// TwinCAT 3 PLC project PLC_SortingSystem_PLC
// libraries:
//   Tc2_MC2, * (Beckhoff Automation GmbH)
//   Tc2_Standard, * (Beckhoff Automation GmbH)
//   Tc2_System, * (Beckhoff Automation GmbH)
//   Tc2_Utilities, * (Beckhoff Automation GmbH)
//   Tc3_Module, * (Beckhoff Automation GmbH)
// project tree:
//   01_Submodules/Axis/ FB_Axis.TcPOU
//   01_Submodules/Cylinder/ITFs/ I_Cylinder.TcIO
//   01_Submodules/Cylinder/POUs/ FB_Cylinder.TcPOU, FB_CylinderDiag.TcPOU, FB_CylinderTemp.TcPOU, FB_CylinderTempDiag.TcPOU, FB_CylinderTempRecord.TcPOU
//   01_Submodules/Signal handling/ITFs/ I_SignalHandling.TcIO
//   01_Submodules/Signal handling/POUs/ FB_SignalHandling.TcPOU, FB_SignalHandlingDelay.TcPOU, FB_SignalHandlingIntern.TcPOU
//   02_Subsystems/ E_StateSeparatingAuto.TcDUT, E_StateSortingAutoAxis.TcDUT, E_StateSortingAutoCylinder.TcDUT, FB_SeparatingModule.TcPOU, FB_SortingModule.TcPOU, FB_Subsystem_Root.TcPOU
//   03_Machine/ E_MachineMode.TcDUT, FB_Machine.TcPOU
//   04_Application/ MAIN.TcPOU
//   00_Internal PackAL/DUTs/ E_PMLState.TcDUT, E_PMLUnitMode.TcDUT
//   00_Internal PackAL/POUs/ PS_PackML_StateMachine_Auto.TcPOU, PS_PackML_StateMachine_Maintenance.TcPOU, PS_PackML_StateMachine_Manual.TcPOU, PS_PackML_StateMachine_SemiAuto.TcPOU, PS_UnitModeManager.TcPOU
//   05_Visu/ FB_Visu.TcPOU, GlobalTextList.TcGTLO, Visu_SortingSystem.TcVIS
//   / PlcTask.TcTTO, Visualization Manager.TcVMO (not stored)

CONFIGURATION PLC_SortingSystem_PLC
    RESOURCE PLC ON TwinCAT3
        TASK PlcTask(INTERVAL := T#10ms, PRIORITY := 20);
        PROGRAM MAIN WITH PlcTask : MAIN;
    END_RESOURCE
END_CONFIGURATION

// ---- 02_Subsystems/E_StateSeparatingAuto.TcDUT
{attribute 'qualified_only'}
{attribute 'strict'}
TYPE E_StateSeparatingAuto :
(
	Init := 0,
	Start,
	CloseClamp,
	OpenBarrier,
	CloseBarrier,
	OpenClamp
);
END_TYPE

// ---- 02_Subsystems/E_StateSortingAutoAxis.TcDUT
{attribute 'qualified_only'}
{attribute 'strict'}
TYPE E_StateSortingAutoAxis :
(
	WaitForCylinderAtWorkPos := 0,
	MoveAxis,
	StopAxis
);
END_TYPE

// ---- 02_Subsystems/E_StateSortingAutoCylinder.TcDUT
{attribute 'qualified_only'}
{attribute 'strict'}
TYPE E_StateSortingAutoCylinder :
(
	DetectBox := 0,
	CylToWork,
	CylToBase
);
END_TYPE

// ---- 03_Machine/E_MachineMode.TcDUT
{attribute 'qualified_only'}
{attribute 'strict'}
TYPE E_MachineMode :
(
	Idle := 0,
	Execute := 1,
	Stopped := 2,
	Aborted := 3,
	Starting := 4,
	Stopping := 5,
	Aborting := 6,
	Resetting := 7
);
END_TYPE

// ---- 00_Internal PackAL/DUTs/E_PMLState.TcDUT
(* states according to PackTags v3.0 *)
{attribute 'qualified_only'}
{attribute 'strict'}
TYPE E_PMLState :
(
	UNDEFINED		:=  0,
	CLEARING 		:=  1,
	STOPPED 		:=  2,
	STARTING 		:=  3,
	IDLE 			:=  4,
	SUSPENDED 		:=  5,
	EXECUTE 		:=  6,
	STOPPING	 	:=  7,
	ABORTING 		:=  8,
	ABORTED 		:=  9,
	HOLDING 		:= 10,
	HELD 			:= 11,
	UNHOLDING 		:= 12,
	SUSPENDING 		:= 13,
	UNSUSPENDING 	:= 14,
	RESETTING 		:= 15,
	COMPLETING 		:= 16,
	COMPLETE	 	:= 17
);
END_TYPE

// ---- 00_Internal PackAL/DUTs/E_PMLUnitMode.TcDUT
{attribute 'qualified_only'}
{attribute 'strict'}
TYPE E_PMLUnitMode :
(
	UNDEFINED		:=  0,
	AUTOMATIC		:=  1,
	MAINTENANCE 	:=  2,
	MANUAL 			:=  3,
	SEMIAUTOMATIC	:=  4,
	DRYRUN			:=  5,
	USERMODE1		:=  6,
	USERMODE2		:=  7,
	IDLE 			:=  8,
	ESTOP 			:=  9
);
END_TYPE

// ---- 01_Submodules/Cylinder/ITFs/I_Cylinder.TcIO
INTERFACE I_Cylinder

PROPERTY bState_AtBasePos : BOOL
GET
END_GET
END_PROPERTY

PROPERTY bState_AtWorkPos : BOOL
GET
END_GET
END_PROPERTY

PROPERTY bState_MoveToWork : BOOL
GET
END_GET
END_PROPERTY

METHOD MoveToBase
VAR_INPUT
END_VAR
END_METHOD

METHOD MoveToWork
VAR_INPUT
END_VAR
END_METHOD

METHOD Reset
VAR_INPUT
END_VAR
END_METHOD

END_INTERFACE

// ---- 01_Submodules/Signal handling/ITFs/I_SignalHandling.TcIO
INTERFACE I_SignalHandling

METHOD PUBLIC Enable
VAR_INPUT
	bEnable		: BOOL;
END_VAR
END_METHOD

METHOD SetOutput
VAR_INPUT
END_VAR
END_METHOD

END_INTERFACE

// ---- 04_Application/MAIN.TcPOU
(* =======================================================================================================================================
   OOP: Extended sample
   =======================================================================================================================================
   Description: 
   This PLC sample contains an object-oriented program to control a sorting system.
   The application can be controlled via an integrated visualization.
   
   PLC_SortingSystem_PLC:
   The functionality of the sorting system is implemented within this PLC project (PLC_SortingSystem_PLC).
   It also contains the visualization to control the application.
   
   PLC_SortingSystem_Simu:
   To run the project without hardware, the simulation PLC can be used.
   For example, It simulates the cylinder positions and temperatures, as well as the sensor signals (correspondent to the box positions). 
   =======================================================================================================================================
   InfoSys:
   https://infosys.beckhoff.de/content/1033/tc3_sampleprogram1/45035996374683915.html?id=6126826020926170206
   https://infosys.beckhoff.de/content/1033/tc3_plc_intro/72057596565231755.html?id=3937754078542861062
   ======================================================================================================================================= *)
PROGRAM MAIN
VAR
	fbMachine						: FB_Machine;
	
	//Added Variables
	Plastic_ActPos			AT %Q* 	: LREAL;
	Plastic_ActVelo			AT %Q* 	: LREAL;
	Metal_ActPos			AT %Q* 	: LREAL;
	Metal_ActVelo			AT %Q* 	: LREAL;
	Separating_ActPos		AT %Q* 	: LREAL;
	Separating_ActVelo		AT %Q* 	: LREAL;
	
	{attribute 'TcAnalytics'}
	eMachineState			AT %Q*	: E_MachineMode;
	
	sNetId	: STRING;
	fbGetLocalNetId	:	FB_GetLocalAmsNetId;
	bBusy	: BOOL;
	bInit	: BOOL;
	
	fbConveyorTimerPlastic			: TON;
	fbConveyorTimerMetal			: TON;
	fbConveyorTimerSeparating		: TON;
	tErrorTime						: TIME := T#60M;	
	
END_VAR

// =========================================================

fbMachine();

// =========================================================

Plastic_ActPos := MAIN.fbMachine.fbPlasticSorting.fbAxis.AxisRef.NcToPlc.ActPos;
Plastic_ActVelo := MAIN.fbMachine.fbPlasticSorting.fbAxis.AxisRef.NcToPlc.ActVelo;

Metal_ActPos := MAIN.fbMachine.fbMetalSorting.fbAxis.AxisRef.NcToPlc.ActPos;
Metal_ActVelo := MAIN.fbMachine.fbMetalSorting.fbAxis.AxisRef.NcToPlc.ActVelo;

Separating_ActPos := MAIN.fbMachine.fbSeparateModule.fbAxis.AxisRef.NcToPlc.ActPos;
Separating_ActVelo := MAIN.fbMachine.fbSeparateModule.fbAxis.AxisRef.NcToPlc.ActVelo;

//Handle Conveyor Threshold Overrun
//IF Separating_ActPos > 10000000 THEN
	
//END_IF

//New Machine Enum

IF fbMachine.fbVisu.bIdle THEN
	eMachineState := 0;
ELSIF NOT fbMachine.fbVisu.bButtonPowerIn THEN
	eMachineState := 3;
ELSIF fbMachine.fbVisu.bStarted THEN
	eMachineState := 1;
ELSIF fbMachine.fbVisu.bStopped THEN
	eMachineState := 2;
ELSIF fbMachine.fbVisu.bButtonStartIn THEN
	eMachineState := 4;
ELSIF fbMachine.fbVisu.bButtonStopIn THEN
	eMachineState := 5;
ELSIF fbMachine.fbVisu.bButtonAbortIn THEN
	eMachineState := 6;
ELSIF fbMachine.fbVisu.bReset THEN
	eMachineState := 7;
END_IF

IF NOT bInit THEN
bInit := GetLocalAmsNetId();
END_IF

METHOD GetLocalAmsNetId : BOOL;
VAR_INPUT
END_VAR
fbGetLocalNetId(
	bExecute:= NOT bBusy, 
	bBusy=> bBusy,
	AddrString=> sNetId);
	
IF NOT ((sNetId = '') OR (sNetId = '0.0.0.0.0.0')) THEN
	GetLocalAmsNetId := TRUE;
	RETURN;
END_IF

GetLocalAmsNetId := FALSE;
RETURN;
END_METHOD

END_PROGRAM

// ---- 03_Machine/FB_Machine.TcPOU
FUNCTION_BLOCK FB_Machine
VAR_INPUT
	// =============== Cylinder choice =========================================================
	// Separating module - Clamp cylinder
	bSeparatingClampDiag				: BOOL := TRUE;							// If true the clamp cylinder has diagnosis functionality
	bSeparatingClampTemp				: BOOL := TRUE;							// If true the clamp cylinder has temperature functionality
	bSeparatingClampRecord				: BOOL := FALSE;						// If true the clamp cylinder has recording functionality
	
	// Separating module - Barrier cylinder
	bSeparatingBarrierDiag 				: BOOL := FALSE;						// If true the barrier cylinder has diagnosis functionality
	bSeparatingBarrierTemp 				: BOOL := TRUE;							// If true the barrier cylinder has temperature functionality
	bSeparatingBarrierRecord			: BOOL := TRUE;							// If true the barrier cylinder has recording functionality
	
	// Sorting module for metal boxes - Cylinder
	bMetalSortingCylinderDiag 			: BOOL := TRUE;							// If true the cylinder for metal boxes has diagnosis functionality
	bMetalSortingCylinderTemp 			: BOOL := TRUE;						// If true the cylinder for metal boxes has temperature functionality
	bMetalSortingCylinderRecord 		: BOOL := FALSE;						// If true the cylinder for metal boxes has recording functionality
	
	// Sorting module for plastic boxes - Cylinder
	bPlasticSortingCylinderDiag 		: BOOL := TRUE;							// If true the cylinder for plastic boxes has diagnosis functionality
	bPlasticSortingCylinderTemp 		: BOOL := TRUE;						// If true the cylinder for plastic boxes has temperature functionality
	bPlasticSortingCylinderRecord 		: BOOL := FALSE;						// If true the cylinder for plastic boxes has recording functionality
	

END_VAR
VAR
//
	fbTimerStop						: TON;
	fStopTimePT						: TIME;
	fStartTimePT					: TIME;
	fbTimerStart					: TON;
	fbDRAND							: DRAND;
	fbTon							: TON;
	iTmrET							: INT;
	fRandom							: LREAL;
	bGenerateNumber					: BOOL := TRUE;	
	iDowntimeCounter				: INT;
	fbTimerDowntime					: TON;
	bDowntime						: BOOL;	
	
	// =============== Varying Package Timing ==============================================
	tPackageTime				: TIME;
	fRandValue					: LREAL;
	fbRand						: DRAND;

	// =============== Error ====================================================================
	bError								: BOOL;									// True if modules have errors
	
	// =============== Axis variable ============================================================
	fAxisVelo							: LREAL;								// Axis velocity
	fAxisVeloLastCycle					: LREAL;								// Axis velocity of last cycle
		
	// =============== State machine variables ==================================================
	bStarted							: BOOL;									// True if state machine is in state EXECUTE
	bStopped							: BOOL;									// True if state machine is in state STOPPED
	bReset						AT %Q*	: BOOL;									// True if state machine is in state RESETTING
	bAborted							: BOOL;									// True if state machine is in state ABORTED
	bIdle								: BOOL;									// True if state machine is in state IDLE
	bAuto								: BOOL;									// True if state machine is in mode AUTOMATIC
	bSemi								: BOOL;									// True if state machine is in mode SEMIAUTOMATIC
	bManual								: BOOL;									// True if state machine is in mode MANUAL
	bMaintenance						: BOOL;									// True if state machine is in mode MAINTENANCE
	bStartButtonOff						: BOOL;									// To turn off start button

	// =============== Machine elements =========================================================
	fbSeparateModule					: FB_SeparatingModule;					// Separating module
	fbMetalSorting						: FB_SortingModule;						// Module that sorts metal boxes
	fbPlasticSorting					: FB_SortingModule;						// Module that sorts plastic boxes
	fbComprAir							: FB_SignalHandlingIntern;				// Compressed air
	fbPowerSupply						: FB_SignalHandlingIntern;				// Power supply
	fbVisu								: FB_Visu;								// Visualization

	// =============== Buttons ==================================================================
	fbButtonStart						: FB_SignalHandlingIntern;				// Button to start the machine
	fbButtonStop						: FB_SignalHandlingIntern;				// Button to stop the machine
	fbButtonReset						: FB_SignalHandlingIntern;				// Button to reset the machine
	fbButtonAbort						: FB_SignalHandlingIntern;				// Button to abort the machine
	fbButtonAuto						: FB_SignalHandlingIntern;				// Button to change machine mode to AUTOMATIC
	fbButtonSemi						: FB_SignalHandlingIntern;				// Button to change machine mode to SEMI-AUTOMATIC
	fbButtonManual						: FB_SignalHandlingIntern;				// Button to change machine mode to MANUAL
	fbButtonMaintenance					: FB_SignalHandlingIntern;				// Button to change machine mode to MAINTENANCE
	fbButtonPower						: FB_SignalHandlingIntern;				// Button to control power supply
	fbButtonComprAir					: FB_SignalHandlingIntern;				// Button to control compressed air

	// =============== State machine ============================================================
	fbStateMachineAuto					: PS_PackML_StateMachine_Auto;			// State machine for mode AUTOMATIC
	fbStateMachineSemiAuto				: PS_PackML_StateMachine_SemiAuto;		// State machine for mode SEMI-AUTOMATIC
	fbStateMachineManual				: PS_PackML_StateMachine_Manual;		// State machine for mode MANUAL
	fbStateMachineMaintenance			: PS_PackML_StateMachine_Maintenance;	// State machine for mode MAINTENANCE
	
	ePMLUnitMode						: E_PMLUnitMode := E_PMLUnitMode.IDLE;	// Current mode
	ePMLUnitModeRequested				: E_PMLUnitMode;						// Requested mode
	fbUnitModeManager					: PS_UnitModeManager;					// Mode manager
	ePMLState					AT %Q*	: E_PMLState := E_PMLState.IDLE;			// Current state
	ePMLStateRequested					: E_PMLState;							// Requested state
	
	// =============== Common variables =========================================================
	bInit								: BOOL;									// True if module parameters are initialized
	bAxisEnable							: BOOL;									// True if it is allowed to move axis
	bManualAxisEnable					: BOOL;									// True if it is allowed to move manually axis
	fbTriggerStart						: R_TRIG;								// To diagnose rising edge of start button
	fbTriggerSeparated					: R_TRIG;								// To diagnose rising edge of separated box
	fbTriggerSelectedM					: R_TRIG;								// To diagnose rising edge of selected metal box
	fbTriggerSelectedP					: R_TRIG;								// To diagnose rising edge of selected plastic box
	nBoxesOnTheWay						: INT;									// Number of boxes being moved
	aClampTemps							: ARRAY[1..100] OF LREAL;				// Temperature of clamp cylinder
	aBarrierTemps						: ARRAY[1..100] OF LREAL;				// Temperature of barrier cylinder
	aMetalTemps							: ARRAY[1..100] OF LREAL;				// Temperature of metal cylinder
	aPlasticTemps						: ARRAY[1..100] OF LREAL;				// Temperature of plastic cylinder
	bStartingIsSetToTrue				: BOOL;									// True if the starting methods were called with input TRUE
	bResetIsSetToTrue					: BOOL;									// True if the resetting methods were called with input TRUE
	bHaltIsSetToTrue					: BOOL;									// True if the halting methods were called with input TRUE
	
	cSeparatingBarrierAtWork			: TIME := T#4.5S;									// Time value for separating process: barrier cylinder stays at work position

END_VAR
VAR CONSTANT
	// =============== Axis velocities ==========================================================
	cAxisVeloAutomatic					: LREAL	:= 100.0;						// Axis velocity in (semi) automatic mode
	cAxisVeloNotAutomatic				: LREAL	:= 50.0;						// Axis velocity in non-automatic mode
	
	// =============== Cylinder parameters for separating module (clamp and barrier cylinder) ===
	cSeparatingTimeOutClamp				: TIME 	:= T#2.5S;						// For clamp cylinder with diagnosis: time in which the cylinder should reach base/work position
	cSeparatingRecordIntervalClamp		: TIME 	:= T#1S;						// Time of intervals to record the temperature of clamp cylinder
	cSeparatingTimeOutBarrier			: TIME 	:= T#3S;						// For barrier cylinder with diagnosis: time in which the cylinder should reach base/work position
	cSeparatingRecordIntervalBarrier	: TIME 	:= T#1S;						// Time of intervals to record the temperature of barrier cylinder
	//cSeparatingBarrierAtWork			: TIME 	:= T#4.5S;						// Time value for separating process: barrier cylinder stays at work position
	
	// =============== Cylinder parameters for sorting module ===================================
	cSortingTimeOutCylinder				: TIME 	:= T#3S;						// For sorting cylinder with diagnosis: time in which the cylinder should reach base/work position
	cSortingRecordInterval				: TIME 	:= T#1S;						// Time of intervals to record the temperature of sorting cylinder
	cSortingMoveAxis					: TIME 	:= T#2.5S;						// Time to move sorting axis
	cSortingSensorDelay					: TIME 	:= T#3S;						// Time to delay signal of sorting sensor
END_VAR

// =========================================================
// Getting errors of modules
	
	bError := fbSeparateModule.bAxisError OR fbSeparateModule.bClampError OR fbSeparateModule.bBarrierError
			OR fbMetalSorting.bAxisError OR fbMetalSorting.bCylError 
			OR fbPlasticSorting.bAxisError OR fbPlasticSorting.bCylError;
	
// =========================================================
// Setting velocities of axes

	IF (ePMLUnitMode = E_PMLUnitMode.AUTOMATIC) OR (ePMLUnitMode = E_PMLUnitMode.SEMIAUTOMATIC) THEN
		fAxisVelo := cAxisVeloAutomatic;
	ELSE
		fAxisVelo := cAxisVeloNotAutomatic;
	END_IF

// =========================================================
// Noticing separated and selected boxes
	
	fbTriggerSeparated(CLK := fbSeparateModule.bSeparated);
	fbTriggerSelectedM(CLK := fbMetalSorting.bSelected);
	fbTriggerSelectedP(CLK := fbPlasticSorting.bSelected);
						
// =========================================================
// Getting cylinder temperatures of modules
	
	aBarrierTemps 	:= fbSeparateModule.aBarrierTemps;
	aClampTemps 	:= fbSeparateModule.aClampTemps;
	aMetalTemps 	:= fbMetalSorting.aTemps;
	aPlasticTemps 	:= fbPlasticSorting.aTemps;

// =========================================================
// Cylinder options of modules - choose desired cylinders with more or less functionality
	
	fbSeparateModule.CylinderOptions(	bClampDiag		:= bSeparatingClampDiag, 
										bClampTemp		:= bSeparatingClampTemp, 
										bClampRecord	:= bSeparatingClampRecord, 
										bBarrierDiag	:= bSeparatingBarrierDiag, 
										bBarrierTemp	:= bSeparatingBarrierTemp, 
										bBarrierRecord	:= bSeparatingBarrierRecord);
	
	fbMetalSorting.CylinderOptions(		bCylinderDiag	:= bMetalSortingCylinderDiag,
										bCylinderTemp	:= bMetalSortingCylinderTemp,
										bCylinderRecord	:= bMetalSortingCylinderRecord);
	
	fbPlasticSorting.CylinderOptions(	bCylinderDiag	:= bPlasticSortingCylinderDiag,
										bCylinderTemp	:= bPlasticSortingCylinderTemp,
										bCylinderRecord	:= bPlasticSortingCylinderRecord);

// =========================================================
// Call of actions

	// Init
	General_Init();

	// Mode and state requests
	General_Requests();
	
	// Enable for power supply, compressed air control and buttons
	General_Enable();
	
	// Input variables of separating and sorting modules
	General_ModuleInputs();
	
	// Output variables
	General_SetOutput();
	
	// State machine
	General_StateMachine();
	
	// Visualization
	General_Visu();

// =========================================================
//Timer to Stop Machine/Restart
IF bGenerateNumber THEN
	fbDRAND(Seed:= 0, Num => fRandom);
	bGenerateNumber := FALSE;
END_IF

//Check if machine powered on 
fStartTimePT := LREAL_TO_TIME(fRandom*100000000);
fStopTimePT := LREAL_TO_TIME(fRandom*20000000);

(*IF fbButtonPower.bInput AND NOT bDowntime THEN
	fbTimerStop(IN := NOT fbTimerStart.Q , PT:= fStartTimePT, Q => , ET =>);
	fbTimerStart(IN := fbTimerStop.Q , PT := fStopTimePT, Q =>, ET =>);
	
	IF fbTimerStop.Q AND bStarted THEN
		bGenerateNumber := TRUE;
		fbButtonStop.bInput := TRUE;
		iDowntimeCounter := iDowntimeCounter + 1;
	END_IF
	
	IF fbTimerStart.Q AND bStopped THEN
		bGenerateNumber := TRUE;
		fbButtonStart.bInput := TRUE;	
	END_IF

	IF bIdle THEN
		fbButtonStart.bInput := TRUE;
	END_IF
END_IF

//Implement planned downtime after 10 ON/OFF cycles
IF (iDowntimeCounter > 20) THEN
	fbButtonStop.bInput := TRUE;
	bDowntime := TRUE;
	IF bStopped THEN
	fbButtonPower.bInput := FALSE;
	END_IF	
END_IF

fbTimerDowntime(IN := NOT fbButtonPower.bInput, PT := T#120M, Q =>, ET =>);

IF fbTimerDowntime.Q THEN
	fbButtonPower.bInput := TRUE;
	iDowntimeCounter := 0;
	bDowntime := FALSE;
END_IF

fbRand(Seed:= 0, Num => fRandValue);

tPackageTime := LREAL_TO_TIME((fRandValue*5000) + 5000);

cSeparatingBarrierAtWork := tPackageTime;*)

METHOD PRIVATE General_Enable
VAR_INPUT
END_VAR
// =========================================================
// Power supply

	fbButtonPower.Enable(bEnable := TRUE);
	fbPowerSupply.Enable(bEnable := TRUE);
	
	fbPowerSupply.bInput := fbButtonPower.bOut;

// =========================================================
// Axis control
								
	IF (ePMLState = E_PMLState.ABORTED) THEN
		bAxisEnable := FALSE;
	ELSIF fbPowerSupply.bOut THEN
		bAxisEnable := TRUE;
	END_IF
	
	bManualAxisEnable := fbPowerSupply.bOut AND (ePMLState = E_PMLState.EXECUTE)
						AND ((ePMLUnitMode = E_PMLUnitMode.MANUAL) OR (ePMLUnitMode = E_PMLUnitMode.MAINTENANCE));
						
// =========================================================
// Compressed air control
	
	IF (ePMLUnitMode <> E_PMLUnitMode.MAINTENANCE) THEN
		fbComprAir.bInput := fbPowerSupply.bOut;
	ELSE
		fbComprAir.bInput := fbButtonComprAir.bOut;
	END_IF
	
	fbComprAir.Enable(bEnable := TRUE);
	fbButtonComprAir.Enable(bEnable := (ePMLUnitMode = E_PMLUnitMode.MAINTENANCE));

// =========================================================
// Enable of separate module

	fbSeparateModule.Enable(bComprAirEnabled	:= fbComprAir.bOut,
							bAxisEnable			:= bAxisEnable,
							bSensorEnable		:= TRUE,
							bManualAxisEnable	:= bManualAxisEnable);

// =========================================================
// Enable of sorting module for metal boxes

	fbMetalSorting.Enable(	bComprAirEnabled	:= fbComprAir.bOut,
							bAxisEnable			:= bAxisEnable,
							bSensorEnable		:= TRUE,
							bManualAxisEnable	:= bManualAxisEnable);

// =========================================================
// Enable of sorting module for plastic boxes

	fbPlasticSorting.Enable(bComprAirEnabled	:= fbComprAir.bOut,
							bAxisEnable			:= bAxisEnable,
							bSensorEnable		:= TRUE,
							bManualAxisEnable	:= bManualAxisEnable);

// =========================================================
// States and modes
		
	// Start button
	fbButtonStart.Enable(bEnable		:= NOT ((ePMLState = E_PMLState.IDLE) AND bError));
	
	// Stop button
	fbButtonStop.Enable(bEnable 		:= (ePMLState = E_PMLState.STOPPING) OR (ePMLState = E_PMLState.EXECUTE) OR (ePMLState = E_PMLState.IDLE));
	
	// Reset button
	fbButtonReset.Enable(bEnable		:= (ePMLState = E_PMLState.STOPPED));
	
	// Abort button
	fbButtonAbort.bInput 				:= NOT fbPowerSupply.bOut;
	
	fbButtonAbort.Enable(bEnable 		:= (ePMLState = E_PMLState.EXECUTE) OR (ePMLState = E_PMLState.STOPPING) OR (ePMLState = E_PMLState.RESETTING));
								
	// Automatic mode button
	fbButtonAuto.Enable(bEnable 		:= (ePMLState = E_PMLState.IDLE) AND (ePMLUnitMode <> E_PMLUnitMode.AUTOMATIC));
	
	// Semi-automatic mode button
	fbButtonSemi.Enable(bEnable 		:= (ePMLState = E_PMLState.IDLE) AND (ePMLUnitMode <> E_PMLUnitMode.SEMIAUTOMATIC));
	
	// Manual mode button
	fbButtonManual.Enable(bEnable 		:= (ePMLState = E_PMLState.IDLE) AND (ePMLUnitMode <> E_PMLUnitMode.MANUAL));
	
	// Maintenance mode button
	fbButtonMaintenance.Enable(bEnable	:= (ePMLState = E_PMLState.IDLE) AND (ePMLUnitMode <> E_PMLUnitMode.MAINTENANCE));

// =========================================================
END_METHOD

METHOD PRIVATE General_Init
VAR_INPUT
END_VAR
// =========================================================

IF NOT bInit THEN
	
	// Time values of separating module
		// Clamp cylinder
		fbSeparateModule.tTimeOutOfClamp 			:= cSeparatingTimeOutClamp;
		fbSeparateModule.tRecordIntervalOfClamp		:= cSeparatingRecordIntervalClamp;
		
		// Barrier cylinder
		fbSeparateModule.tTimeOutOfBarrier 			:= cSeparatingTimeOutBarrier;
		fbSeparateModule.tRecordIntervalOfBarrier 	:= cSeparatingRecordIntervalBarrier;
		
		// Separating process
		fbSeparateModule.tBarrierAtWorkPos				:= cSeparatingBarrierAtWork;

	// Time values of sorting module (metal boxes)
		fbMetalSorting.tTimeOutOfCylinder 			:= cSortingTimeOutCylinder;
		fbMetalSorting.tRecordIntervalOfCylinder 	:= cSortingRecordInterval;
		fbMetalSorting.tAxisMovement 				:= cSortingMoveAxis;
		fbMetalSorting.tDelayOfSensor 				:= cSortingSensorDelay;
		
	// Time values of sorting module (plastic boxes)
		fbPlasticSorting.tTimeOutOfCylinder 		:= cSortingTimeOutCylinder;
		fbPlasticSorting.tRecordIntervalOfCylinder := cSortingRecordInterval;
		fbPlasticSorting.tAxisMovement 				:= cSortingMoveAxis;
		fbPlasticSorting.tDelayOfSensor 			:= cSortingSensorDelay;

	// Init done
		bInit := TRUE;
END_IF

// =========================================================
END_METHOD

METHOD PRIVATE General_ModuleInputs
VAR_INPUT
END_VAR
// =========================================================
// Separating modul

	// Sate and button signals
	fbSeparateModule.bExecute 			:= (ePMLState = E_PMLState.EXECUTE);
	fbSeparateModule.bSemiStart 		:= fbTriggerStart.Q;
	
	// Axis velocity has changed
	IF (fAxisVeloLastCycle <> fAxisVelo) THEN
		fbSeparateModule.fAxisVelocity 	:= fAxisVelo;
	END_IF
	
	// Information about number of boxes being sorted
	fbSeparateModule.nBoxesOnTheWay 	:= nBoxesOnTheWay;

// =========================================================
// Sorting modul for metal boxes
	
	// Axis velocity has changed
	IF (fAxisVeloLastCycle <> fAxisVelo) THEN
		fbMetalSorting.fAxisVelocity 	:= fAxisVelo;
	END_IF

// =========================================================
// Sorting modul for plastic boxes

	// Axis velocity has changed
	IF (fAxisVeloLastCycle <> fAxisVelo) THEN
		fbPlasticSorting.fAxisVelocity 	:= fAxisVelo;
	END_IF
	
// =========================================================
/// Remember axis velocity of this cycle for next cycle => call of property AxisVelocity is event triggered

	fAxisVeloLastCycle := fAxisVelo;

// =========================================================
END_METHOD

METHOD PRIVATE General_Requests
VAR_INPUT
END_VAR
// =========================================================
// Check for state requests

	fbTriggerStart( CLK := fbButtonStart.bOut);
	
	IF bStartButtonOff AND NOT fbButtonStart.bInput THEN
		bStartButtonOff := FALSE;
	END_IF
	
	IF fbTriggerStart.Q THEN
		bStartButtonOff := TRUE;
	
		IF ePMLState = E_PMLState.ABORTED THEN
			ePMLStateRequested := E_PMLState.CLEARING;
			
		ELSIF ePMLState = E_PMLState.STOPPED THEN
			ePMLStateRequested := E_PMLState.RESETTING;
			
		ELSIF ePMLState = E_PMLState.IDLE AND fbPowerSupply.bOut THEN
			ePMLStateRequested := E_PMLState.STARTING;
		END_IF
		
	ELSIF fbButtonStop.bOut THEN
		ePMLStateRequested := E_PMLState.STOPPING;
		
	ELSIF fbButtonReset.bOut THEN
		ePMLStateRequested := E_PMLState.RESETTING;
	END_IF

// =========================================================
// Check for mode requests

	IF fbButtonManual.bOut THEN
		ePMLUnitModeRequested := E_PMLUnitMode.MANUAL;
		
	ELSIF fbButtonAuto.bOut THEN
		ePMLUnitModeRequested := E_PMLUnitMode.AUTOMATIC;
		
	ELSIF fbButtonSemi.bOut THEN
		ePMLUnitModeRequested := E_PMLUnitMode.SEMIAUTOMATIC;
		
	ELSIF fbButtonMaintenance.bOut THEN
		ePMLUnitModeRequested := E_PMLUnitMode.MAINTENANCE;
	END_IF
	
	IF fbButtonManual.bOut OR fbButtonAuto.bOut OR fbButtonSemi.bOut OR fbButtonMaintenance.bOut THEN
		fbUnitModeManager(	Execute 		:= TRUE,
							eModeCommand 	:= ePMLUnitModeRequested,
							ePMLState 		:= ePMLState);
	END_IF
	
	IF fbUnitModeManager.Done THEN
		ePMLUnitMode := fbUnitModeManager.eModeStatus;
		
		fbUnitModeManager(Execute := FALSE);
	END_IF
	
// =========================================================
END_METHOD

METHOD PRIVATE General_SetOutput
VAR_INPUT
END_VAR
// =========================================================
// State variables

	bStopped 		:= (ePMLState = E_PMLState.STOPPED);
	bStarted 		:= (ePMLState = E_PMLState.EXECUTE);
	bReset 			:= (ePMLState = E_PMLState.RESETTING);
	bAborted 		:= (ePMLState = E_PMLState.ABORTED);
	bIdle 			:= (ePMLState = E_PMLState.IDLE AND fbPowerSupply.bOut);

// =========================================================
// Mode variables

	bAuto 			:= (ePMLUnitMode = E_PMLUnitMode.AUTOMATIC);
	bSemi 			:= (ePMLUnitMode = E_PMLUnitMode.SEMIAUTOMATIC);
	bManual 		:= (ePMLUnitMode = E_PMLUnitMode.MANUAL);
	bMaintenance 	:= (ePMLUnitMode = E_PMLUnitMode.MAINTENANCE);

// =========================================================
// Power supply and compressed air control
		
	fbPowerSupply.SetOutput();
	fbComprAir.SetOutput();		

// =========================================================
// Modules

	fbSeparateModule.InputOutput();
	fbMetalSorting.InputOutput();
	fbPlasticSorting.InputOutput();

// =========================================================
// Buttons

	// Power supply and compressed air control
	fbButtonPower.SetOutput();
	fbButtonComprAir.SetOutput();	
	
	// States
	fbButtonStart.SetOutput();
	fbButtonStop.SetOutput();
	fbButtonReset.SetOutput();
	fbButtonAbort.SetOutput();
	
	// Modes
	fbButtonAuto.SetOutput();
	fbButtonSemi.SetOutput();
	fbButtonManual.SetOutput();
	fbButtonMaintenance.SetOutput();	
	
// =========================================================
END_METHOD

METHOD PRIVATE General_StateMachine
VAR_INPUT
END_VAR
// =========================================================
	// Mode and state handling
	
CASE ePMLUnitMode OF
	
	// =========================================================	
	E_PMLUnitMode.AUTOMATIC:		

				fbStateMachineAuto(	Start 	:= ePMLStateRequested = E_PMLState.STARTING,
									Stop 	:= fbButtonStop.bOut,
									Reset 	:= fbButtonReset.bOut OR ePMLStateRequested = E_PMLState.RESETTING,
									Clear 	:= ePMLStateRequested = E_PMLState.CLEARING,
									Abort 	:= fbButtonAbort.bOut OR (bError AND ePMLState = E_PMLState.EXECUTE));
								 
				ePMLState := fbStateMachineAuto.ePMLState;
				
				Operating_Automatic();

	// =========================================================	
	E_PMLUnitMode.MANUAL:		

				fbStateMachineManual(	Start 	:= ePMLStateRequested = E_PMLState.STARTING,
										Stop 	:= fbButtonStop.bOut,
										Reset 	:= fbButtonReset.bOut OR ePMLStateRequested = E_PMLState.RESETTING,
										Clear 	:= ePMLStateRequested = E_PMLState.CLEARING,
										Abort 	:= fbButtonAbort.bOut OR (bError AND ePMLState = E_PMLState.EXECUTE));
									 
				ePMLState := fbStateMachineManual.ePMLState;
				
				Operating_Manual();
	
	// =========================================================						
	E_PMLUnitMode.SEMIAUTOMATIC:	

				fbStateMachineSemiAuto(	Start 	:= ePMLStateRequested = E_PMLState.STARTING,
									 	Stop 	:= fbButtonStop.bOut,
										Reset 	:= fbButtonReset.bOut OR ePMLStateRequested = E_PMLState.RESETTING,
										Clear 	:= ePMLStateRequested = E_PMLState.CLEARING,
										Abort 	:= fbButtonAbort.bOut OR (bError AND ePMLState = E_PMLState.EXECUTE));
									 
				ePMLState := fbStateMachineSemiAuto.ePMLState;
				
				Operating_Semiautomatic();
	
	// =========================================================						
	E_PMLUnitMode.MAINTENANCE:	

				fbStateMachineMaintenance(	Start 	:= ePMLStateRequested = E_PMLState.STARTING,
											Stop 	:= fbButtonStop.bOut,
											Reset 	:= fbButtonReset.bOut OR ePMLStateRequested = E_PMLState.RESETTING,
											Clear 	:= ePMLStateRequested = E_PMLState.CLEARING,
											Abort 	:= fbButtonAbort.bOut OR (bError AND ePMLState = E_PMLState.EXECUTE));
									 
				ePMLState := fbStateMachineMaintenance.ePMLState;
				
				Operating_Maintenance();
END_CASE

// =========================================================
END_METHOD

METHOD PRIVATE General_Visu
VAR_INPUT
END_VAR
// =========================================================
		// Calling visu function block
		
fbVisu(	bError  				:= bError, 
		fAxisVelo 				:= fAxisVelo, 
		bComprAirEnabled 		:= fbComprAir.bOut, 
		bPowerEnabled 			:= fbPowerSupply.bOut, 
		bMainAxisMoves 			:= fbSeparateModule.bAxisMoves, 
		bMetalAxisMoves 		:= fbMetalSorting.bAxisMoves, 
		bPlasticAxisMoves 		:= fbPlasticSorting.bAxisMoves, 
		bClampToWork 			:= fbSeparateModule.bClampToWork, 
		bBarrierToWork 			:= fbSeparateModule.bBarrierToWork, 
		bMetalToWork 			:= fbMetalSorting.bCylinderToWork, 
		bPlasticToWork 			:= fbPlasticSorting.bCylinderToWork, 
		bClampError 			:= fbSeparateModule.bClampError, 
		sClampErrMsg 			:= fbSeparateModule.sClampErrorMsg, 
		bMetalCylError 			:= fbMetalSorting.bCylError, 
		sMetalErrMsg 			:= fbMetalSorting.sCylErrorMsg, 
		bPlasticCylError 		:= fbPlasticSorting.bCylError, 
		sPlasticErrMsg 			:= fbPlasticSorting.sCylErrorMsg, 
		nMainAxisErrorId 		:= fbSeparateModule.fbAxis.nErrorID, 
		nMetalAxisErrorId 		:= fbMetalSorting.fbAxis.nErrorID, 
		nPlasticAxisErrorId		:= fbPlasticSorting.fbAxis.nErrorID, 
		bStarted 				:= bStarted, 
		bStopped 				:= bStopped, 
		bReset 					:= bReset, 
		bAborted 				:= bAborted, 
		bIdle					:= bIdle, 
		bAuto 					:= bAuto, 
		bSemi 					:= bSemi, 
		bManual 				:= bManual, 
		bMaintenance 			:= bMaintenance, 
		bStartButtonOff 		:= bStartButtonOff, 
		bButtonPowerIn 			:= fbButtonPower.bOut, 
		bButtonComprAirIn 		:= fbButtonComprAir.bOut, 
		bButtonStartIn 			:= fbButtonStart.bOut, 
		bButtonStopIn 			:= fbButtonStop.bOut, 
		bButtonResetIn 			:= fbButtonReset.bOut, 
		bButtonAbortIn 			:= fbButtonAbort.bOut, 
		bButtonAutoIn 			:= fbButtonAuto.bOut, 
		bButtonSemiIn 			:= fbButtonSemi.bOut, 
		bButtonManuIn 			:= fbButtonManual.bOut, 
		bButtonMaintenanceIn 	:= fbButtonMaintenance.bOut, 
		bButtonMainFwIn 		:= fbSeparateModule.bButtonAxisFwOut,
		bButtonMainBwIn 		:= fbSeparateModule.bButtonAxisBwOut, 
		bButtonMetalFwIn 		:= fbMetalSorting.bButtonAxisFwOut, 
		bButtonMetalBwIn 		:= fbMetalSorting.bButtonAxisBwOut, 
		bButtonPlasticFwIn 		:= fbPlasticSorting.bButtonAxisFwOut, 
		bButtonPlasticBwIn 		:= fbPlasticSorting.bButtonAxisBwOut, 
		bButtonClampToWorkIn 	:= fbSeparateModule.bButtonClampToWorkOut, 
		bButtonBarrierToWorkIn 	:= fbSeparateModule.bButtonBarrierToWorkOut, 
		bButtonMetalToWorkIn 	:= fbMetalSorting.bButtonCylToWorkOut, 
		bButtonPlasticToWorkIn 	:= fbPlasticSorting.bButtonCylToWorkOut, 
		
		bButtonPowerOut			=> fbButtonPower.bInput, 
		bButtonComprAirOut 		=> fbButtonComprAir.bInput, 
		bButtonStartOut 		=> fbButtonStart.bInput, 
		bButtonStopOut 			=> fbButtonStop.bInput, 
		bButtonResetOut 		=> fbButtonReset.bInput, 
		bButtonAutoOut 			=> fbButtonAuto.bInput, 
		bButtonSemiOut 			=> fbButtonSemi.bInput, 
		bButtonManuOut 			=> fbButtonManual.bInput, 
		bButtonMaintenanceOut 	=> fbButtonMaintenance.bInput, 
		bButtonMainFwOut 		=> fbSeparateModule.bButtonAxisFwIn, 
		bButtonMainBwOut 		=> fbSeparateModule.bButtonAxisBwIn, 
		bButtonMetalFwOut 		=> fbMetalSorting.bButtonAxisFwIn, 
		bButtonMetalBwOut 		=> fbMetalSorting.bButtonAxisBwIn, 
		bButtonPlasticFwOut		=> fbPlasticSorting.bButtonAxisFwIn, 
		bButtonPlasticBwOut		=> fbPlasticSorting.bButtonAxisBwIn, 
		bButtonClampToWorkOut 	=> fbSeparateModule.bButtonClampToWorkIn, 
		bButtonBarrierToWorkOut	=> fbSeparateModule.bButtonBarrierToWorkIn, 
		bButtonMetalToWorkOut 	=> fbMetalSorting.bButtonCylToWorkIn, 
		bButtonPlasticToWorkOut	=> fbPlasticSorting.bButtonCylToWorkIn);
	
// =========================================================
END_METHOD

METHOD PRIVATE Operating_Automatic
VAR_INPUT
END_VAR
// =========================================================

CASE ePMLState OF
	
	// =========================================================
	// Turning axis reset off, passing it to axis instances
	E_PMLState.IDLE:
	
				IF bResetIsSetToTrue THEN
					bResetIsSetToTrue := FALSE;
					
					fbSeparateModule.Reset(bReset := FALSE);							
					fbMetalSorting.Reset(bReset := FALSE);
					fbPlasticSorting.Reset(bReset := FALSE);
					
					fbStateMachineAuto.StateComplete := FALSE;	
				END_IF
	
	// =========================================================
	// Resetting variables for executing automatic mode, checking status of axes
	E_PMLState.STARTING:
	
				IF NOT bStartingIsSetToTrue THEN
					bStartingIsSetToTrue := TRUE;
					
					fbSeparateModule.Starting(bStarting := TRUE);
					fbMetalSorting.Starting(bStarting := TRUE);
					fbPlasticSorting.Starting(bStarting := TRUE);
				END_IF

				IF NOT fbSeparateModule.bState_StartingDone THEN
					fbSeparateModule.Starting(bStarting := TRUE);
				END_IF
				
				IF NOT fbMetalSorting.bState_StartingDone THEN
					fbMetalSorting.Starting(bStarting := TRUE);
				END_IF
				
				IF NOT fbPlasticSorting.bState_StartingDone THEN
					fbPlasticSorting.Starting(bStarting := TRUE);
				END_IF

				IF fbSeparateModule.bState_StartingDone AND fbMetalSorting.bState_StartingDone AND fbPlasticSorting.bState_StartingDone THEN
					fbStateMachineAuto.StateComplete := TRUE;
				END_IF

	// =========================================================
	// Executing automatic mode
	E_PMLState.EXECUTE:	

				IF bStartingIsSetToTrue THEN
					bStartingIsSetToTrue := FALSE;
					
					fbSeparateModule.Starting(bStarting := FALSE);
					fbMetalSorting.Starting(bStarting := FALSE);	
					fbPlasticSorting.Starting(bStarting := FALSE);
					
					fbStateMachineAuto.StateComplete := FALSE;
				END_IF
				
				fbSeparateModule.Automatic();
				fbMetalSorting.Automatic();
				fbPlasticSorting.Automatic();
				
				IF fbTriggerSeparated.Q THEN
					nBoxesOnTheWay := nBoxesOnTheWay + 1;
				END_IF
				
				IF fbTriggerSelectedM.Q THEN
					nBoxesOnTheWay := nBoxesOnTheWay - 1;
				END_IF
				
				IF fbTriggerSelectedP.Q THEN
					nBoxesOnTheWay := nBoxesOnTheWay - 1;
				END_IF
						
	// =========================================================
	// Stopping axes
	E_PMLState.ABORTING:

				IF NOT bHaltIsSetToTrue THEN
					bHaltIsSetToTrue := TRUE;
					
					fbSeparateModule.Stop(bHalt := TRUE);
					fbMetalSorting.Stop(bHalt := TRUE);
					fbPlasticSorting.Stop(bHalt := TRUE);
				END_IF

				IF NOT fbSeparateModule.bState_HaltDone THEN
					fbSeparateModule.Stop(bHalt := TRUE);
				END_IF
				
				IF NOT fbMetalSorting.bState_HaltDone THEN
					fbMetalSorting.Stop(bHalt := TRUE);
				END_IF
				
				IF NOT fbPlasticSorting.bState_HaltDone THEN
					fbPlasticSorting.Stop(bHalt := TRUE);
				END_IF

				IF fbSeparateModule.bState_HaltDone AND fbMetalSorting.bState_HaltDone AND fbPlasticSorting.bState_HaltDone THEN
					fbStateMachineAuto.StateComplete := TRUE;
				END_IF
	
	// =========================================================
	// Turning off axis stop, passing it to axis instances
	E_PMLState.ABORTED:
				
				IF bHaltIsSetToTrue THEN
					bHaltIsSetToTrue := FALSE;
					
					fbSeparateModule.Stop(bHalt := FALSE);
					fbMetalSorting.Stop(bHalt := FALSE);
					fbPlasticSorting.Stop(bHalt := FALSE);
				END_IF
				
				IF fbStateMachineAuto.StateComplete THEN
					fbStateMachineAuto.StateComplete := FALSE;
				END_IF
	
	// =========================================================
	E_PMLState.CLEARING:

				fbStateMachineAuto.StateComplete := TRUE;
	
	// =========================================================
	// Selecting boxes on conveyor belt to destination, then stopping axes
	E_PMLState.STOPPING:	

				IF fbTriggerSeparated.Q THEN
					nBoxesOnTheWay := nBoxesOnTheWay + 1;
				END_IF
				
				IF fbTriggerSelectedM.Q THEN
					nBoxesOnTheWay := nBoxesOnTheWay - 1;
				END_IF
				
				IF fbTriggerSelectedP.Q THEN
					nBoxesOnTheWay := nBoxesOnTheWay - 1;
				END_IF
				
				IF (nBoxesOnTheWay = 0) AND NOT bHaltIsSetToTrue THEN
					bHaltIsSetToTrue := TRUE;
		
					fbSeparateModule.Stop(bHalt := TRUE);				
					fbMetalSorting.Stop(bHalt := TRUE);				
					fbPlasticSorting.Stop(bHalt := TRUE);			
				END_IF
				
				IF NOT fbSeparateModule.bState_HaltDone OR (nBoxesOnTheWay <> 0) THEN
					fbSeparateModule.Automatic();
					
					IF (nBoxesOnTheWay = 0) THEN
						fbSeparateModule.Stop(bHalt := TRUE);
					END_IF
				END_IF
				
				IF NOT fbMetalSorting.bState_HaltDone OR (nBoxesOnTheWay <> 0) THEN
					fbMetalSorting.Automatic();
					
					IF (nBoxesOnTheWay = 0) THEN
						fbMetalSorting.Stop(bHalt := TRUE);
					END_IF
				END_IF
				
				IF NOT fbPlasticSorting.bState_HaltDone OR (nBoxesOnTheWay <> 0) THEN
					fbPlasticSorting.Automatic();
					
					IF (nBoxesOnTheWay = 0) THEN
						fbPlasticSorting.Stop(bHalt := TRUE);
					END_IF
				END_IF

				IF fbSeparateModule.bState_HaltDone AND fbMetalSorting.bState_HaltDone
				AND fbPlasticSorting.bState_HaltDone AND (nBoxesOnTheWay = 0) THEN
					fbStateMachineAuto.StateComplete := TRUE;
				END_IF
					
	// =========================================================
	// Turning off axis stop, passing it to axis instances
	E_PMLState.STOPPED:	

				IF bHaltIsSetToTrue THEN
					bHaltIsSetToTrue := FALSE;
					
					fbSeparateModule.Stop(bHalt := FALSE);	
					fbMetalSorting.Stop(bHalt := FALSE);			
					fbPlasticSorting.Stop(bHalt := FALSE);
				END_IF

				IF fbStateMachineAuto.StateComplete THEN
					fbStateMachineAuto.StateComplete := FALSE;	
				END_IF

	// =========================================================
	// Resetting cylinders and axes
	E_PMLState.RESETTING:	

				IF NOT bResetIsSetToTrue THEN
					bResetIsSetToTrue := TRUE;
					
					fbSeparateModule.Reset(bReset := TRUE);							
					fbMetalSorting.Reset(bReset := TRUE);
					fbPlasticSorting.Reset(bReset := TRUE);
				END_IF
				
				IF NOT fbSeparateModule.bState_ResetDone THEN
					fbSeparateModule.Reset(bReset := TRUE);
				END_IF
				
				IF NOT fbMetalSorting.bState_ResetDone THEN
					fbMetalSorting.Reset(bReset := TRUE);
				END_IF
				
				IF NOT fbPlasticSorting.bState_ResetDone THEN
					fbPlasticSorting.Reset(bReset := TRUE);
				END_IF
				
				IF fbSeparateModule.bState_ResetDone AND fbMetalSorting.bState_ResetDone AND fbPlasticSorting.bState_ResetDone 
				AND fbSeparateModule.bState_ClampAtBasePos AND fbSeparateModule.bState_BarrierAtBasePos
				AND fbMetalSorting.bState_CylinderAtBasePos AND fbPlasticSorting.bState_CylinderAtBasePos THEN
					nBoxesOnTheWay 						:= 0;
					fbStateMachineAuto.StateComplete 	:= TRUE;
				END_IF
END_CASE

// =========================================================
END_METHOD

METHOD PRIVATE Operating_Maintenance
VAR_INPUT
END_VAR
// =========================================================

CASE ePMLState OF
	
	// =========================================================
	// Turning axis reset off, passing it to axis instances
	E_PMLState.IDLE:		

				IF bResetIsSetToTrue THEN
					bResetIsSetToTrue := FALSE;
					
					fbSeparateModule.Reset(bReset := FALSE);
					fbMetalSorting.Reset(bReset := FALSE);
					fbPlasticSorting.Reset(bReset := FALSE);
					
					fbStateMachineMaintenance.StateComplete := FALSE;
				END_IF
	
	// =========================================================
	// Checking status of axes
	E_PMLState.STARTING:	

				IF NOT bStartingIsSetToTrue THEN
					bStartingIsSetToTrue := TRUE;
					
					fbSeparateModule.Starting(bStarting := TRUE);
					fbMetalSorting.Starting(bStarting := TRUE);
					fbPlasticSorting.Starting(bStarting := TRUE);
				END_IF

				IF NOT fbSeparateModule.bState_StartingDone THEN
					fbSeparateModule.Starting(bStarting := TRUE);
				END_IF
				
				IF NOT fbMetalSorting.bState_StartingDone THEN
					fbMetalSorting.Starting(bStarting := TRUE);
				END_IF
				
				IF NOT fbPlasticSorting.bState_StartingDone THEN
					fbPlasticSorting.Starting(bStarting := TRUE);
				END_IF

				IF fbSeparateModule.bState_StartingDone AND fbMetalSorting.bState_StartingDone AND fbPlasticSorting.bState_StartingDone THEN
					fbStateMachineMaintenance.StateComplete := TRUE;
				END_IF

	// =========================================================
	// Executing maintenance mode
	E_PMLState.EXECUTE:	

				IF bStartingIsSetToTrue THEN
					bStartingIsSetToTrue := FALSE;
					
					fbSeparateModule.Starting(bStarting := FALSE);
					fbMetalSorting.Starting(bStarting := FALSE);	
					fbPlasticSorting.Starting(bStarting := FALSE);
					
					fbStateMachineMaintenance.StateComplete := FALSE;
				END_IF
				
				fbSeparateModule.Maintenance();
				fbMetalSorting.Maintenance();
				fbPlasticSorting.Maintenance();
						
	// =========================================================
	// Stopping axes
	E_PMLState.ABORTING:	

				IF NOT bHaltIsSetToTrue THEN
					bHaltIsSetToTrue := TRUE;
					
					fbSeparateModule.Stop(bHalt := TRUE);
					fbMetalSorting.Stop(bHalt := TRUE);
					fbPlasticSorting.Stop(bHalt := TRUE);
				END_IF

				IF NOT fbSeparateModule.bState_HaltDone THEN
					fbSeparateModule.Stop(bHalt := TRUE);
				END_IF
				
				IF NOT fbMetalSorting.bState_HaltDone THEN
					fbMetalSorting.Stop(bHalt := TRUE);
				END_IF
				
				IF NOT fbPlasticSorting.bState_HaltDone THEN
					fbPlasticSorting.Stop(bHalt := TRUE);
				END_IF

				IF fbSeparateModule.bState_HaltDone AND fbMetalSorting.bState_HaltDone AND fbPlasticSorting.bState_HaltDone THEN
					fbStateMachineMaintenance.StateComplete := TRUE;
				END_IF
	
	// =========================================================
	// Turning off axis stop, passing it to axis instances
	E_PMLState.ABORTED:	

				IF bHaltIsSetToTrue THEN
					bHaltIsSetToTrue := FALSE;
					
					fbSeparateModule.Stop(bHalt := FALSE);
					fbMetalSorting.Stop(bHalt := FALSE);
					fbPlasticSorting.Stop(bHalt := FALSE);
				END_IF

				IF fbStateMachineMaintenance.StateComplete THEN
					fbStateMachineMaintenance.StateComplete := FALSE;
				END_IF
	
	// =========================================================
	E_PMLState.CLEARING:	

				fbStateMachineMaintenance.StateComplete := TRUE;
	
	// =========================================================
	// Stopping axes
	E_PMLState.STOPPING:	

				IF NOT bHaltIsSetToTrue THEN
					bHaltIsSetToTrue := TRUE;

					fbSeparateModule.Stop(bHalt := TRUE);				
					fbMetalSorting.Stop(bHalt := TRUE);				
					fbPlasticSorting.Stop(bHalt := TRUE);				
				END_IF

				IF NOT fbSeparateModule.bState_HaltDone THEN
					fbSeparateModule.Stop(bHalt := TRUE);
				END_IF
				
				IF NOT fbMetalSorting.bState_HaltDone THEN
					fbMetalSorting.Stop(bHalt := TRUE);
				END_IF
				
				IF NOT fbPlasticSorting.bState_HaltDone THEN
					fbPlasticSorting.Stop(bHalt := TRUE);
				END_IF

				IF fbSeparateModule.bState_HaltDone AND fbMetalSorting.bState_HaltDone AND fbPlasticSorting.bState_HaltDone THEN
						fbStateMachineMaintenance.StateComplete := TRUE;
				END_IF
					
	// =========================================================
	// Turning off axis stop, passing it to axis instances
	E_PMLState.STOPPED:	

				IF bHaltIsSetToTrue THEN
					bHaltIsSetToTrue := FALSE;
					
					fbSeparateModule.Stop(bHalt := FALSE);	
					fbMetalSorting.Stop(bHalt := FALSE);			
					fbPlasticSorting.Stop(bHalt := FALSE);
				END_IF

				IF fbStateMachineMaintenance.StateComplete THEN
					fbStateMachineMaintenance.StateComplete := FALSE;
				END_IF

	// =========================================================
	// Resetting cylinders and axes
	E_PMLState.RESETTING:	

				IF NOT bResetIsSetToTrue THEN
					bResetIsSetToTrue := TRUE;
					
					fbSeparateModule.Reset(bReset := TRUE);							
					fbMetalSorting.Reset(bReset := TRUE);
					fbPlasticSorting.Reset(bReset := TRUE);
				END_IF
				
				IF NOT fbSeparateModule.bState_ResetDone THEN
					fbSeparateModule.Reset(bReset := TRUE);
				END_IF
				
				IF NOT fbMetalSorting.bState_ResetDone THEN
					fbMetalSorting.Reset(bReset := TRUE);
				END_IF
				
				IF NOT fbPlasticSorting.bState_ResetDone THEN
					fbPlasticSorting.Reset(bReset := TRUE);
				END_IF
				
				IF fbSeparateModule.bState_ResetDone AND fbMetalSorting.bState_ResetDone AND fbPlasticSorting.bState_ResetDone 
				AND fbSeparateModule.bState_ClampAtBasePos AND fbSeparateModule.bState_BarrierAtBasePos
				AND fbMetalSorting.bState_CylinderAtBasePos AND fbPlasticSorting.bState_CylinderAtBasePos THEN
					fbStateMachineMaintenance.StateComplete := TRUE;
				END_IF
END_CASE

// =========================================================
END_METHOD

METHOD PRIVATE Operating_Manual
VAR_INPUT
END_VAR
// =========================================================

CASE ePMLState OF
	
	// =========================================================
	// Turning axis reset off, passing it to axis instances
	E_PMLState.IDLE:		

				IF bResetIsSetToTrue THEN
					bResetIsSetToTrue := FALSE;
					
					fbSeparateModule.Reset(bReset := FALSE);
					fbMetalSorting.Reset(bReset := FALSE);
					fbPlasticSorting.Reset(bReset := FALSE);
					
					fbStateMachineManual.StateComplete := FALSE;
				END_IF
	
	// =========================================================
	// Checking status of axes
	E_PMLState.STARTING:	

				IF NOT bStartingIsSetToTrue THEN
					bStartingIsSetToTrue := TRUE;
					
					fbSeparateModule.Starting(bStarting := TRUE);
					fbMetalSorting.Starting(bStarting := TRUE);
					fbPlasticSorting.Starting(bStarting := TRUE);
				END_IF

				IF NOT fbSeparateModule.bState_StartingDone THEN
					fbSeparateModule.Starting(bStarting := TRUE);
				END_IF
				
				IF NOT fbMetalSorting.bState_StartingDone THEN
					fbMetalSorting.Starting(bStarting := TRUE);
				END_IF
				
				IF NOT fbPlasticSorting.bState_StartingDone THEN
					fbPlasticSorting.Starting(bStarting := TRUE);
				END_IF

				IF fbSeparateModule.bState_StartingDone AND fbMetalSorting.bState_StartingDone AND fbPlasticSorting.bState_StartingDone THEN
					fbStateMachineManual.StateComplete := TRUE;
				END_IF

	// =========================================================
	// Executing manual mode
	E_PMLState.EXECUTE:	

				IF bStartingIsSetToTrue THEN
					bStartingIsSetToTrue := FALSE;
					
					fbSeparateModule.Starting(bStarting := FALSE);
					fbMetalSorting.Starting(bStarting := FALSE);
					fbPlasticSorting.Starting(bStarting := FALSE);
					
					fbStateMachineManual.StateComplete := FALSE;
				END_IF
				
				fbSeparateModule.Manual();
				fbMetalSorting.Manual();
				fbPlasticSorting.Manual();
						
	// =========================================================
	// Stopping axes
	E_PMLState.ABORTING:	

				IF NOT bHaltIsSetToTrue THEN
					bHaltIsSetToTrue := TRUE;
					
					fbSeparateModule.Stop(bHalt := TRUE);
					fbMetalSorting.Stop(bHalt := TRUE);
					fbPlasticSorting.Stop(bHalt := TRUE);
				END_IF

				IF NOT fbSeparateModule.bState_HaltDone THEN
					fbSeparateModule.Stop(bHalt := TRUE);
				END_IF
				
				IF NOT fbMetalSorting.bState_HaltDone THEN
					fbMetalSorting.Stop(bHalt := TRUE);
				END_IF
				
				IF NOT fbPlasticSorting.bState_HaltDone THEN
					fbPlasticSorting.Stop(bHalt := TRUE);
				END_IF

				IF fbSeparateModule.bState_HaltDone AND fbMetalSorting.bState_HaltDone AND fbPlasticSorting.bState_HaltDone THEN
					fbStateMachineManual.StateComplete := TRUE;
				END_IF
	
	// =========================================================
	// Turning off axis stop, passing it to axis instances
	E_PMLState.ABORTED:	

				IF bHaltIsSetToTrue THEN
					bHaltIsSetToTrue := FALSE;
					
					fbSeparateModule.Stop(bHalt := FALSE);
					fbMetalSorting.Stop(bHalt := FALSE);
					fbPlasticSorting.Stop(bHalt := FALSE);
				END_IF

				IF fbStateMachineManual.StateComplete THEN
					fbStateMachineManual.StateComplete := FALSE;
				END_IF
	
	// =========================================================
	E_PMLState.CLEARING:	

				fbStateMachineManual.StateComplete := TRUE;
	
	// =========================================================
	// Stopping axes
	E_PMLState.STOPPING:	

				IF NOT bHaltIsSetToTrue THEN
					bHaltIsSetToTrue := TRUE;
					
					fbSeparateModule.Stop(bHalt := TRUE);				
					fbMetalSorting.Stop(bHalt := TRUE);				
					fbPlasticSorting.Stop(bHalt := TRUE);	
				END_IF

				IF NOT fbSeparateModule.bState_HaltDone THEN
					fbSeparateModule.Stop(bHalt := TRUE);
				END_IF
				
				IF NOT fbMetalSorting.bState_HaltDone THEN
					fbMetalSorting.Stop(bHalt := TRUE);
				END_IF
				
				IF NOT fbPlasticSorting.bState_HaltDone THEN
					fbPlasticSorting.Stop(bHalt := TRUE);
				END_IF

				IF fbSeparateModule.bState_HaltDone AND fbMetalSorting.bState_HaltDone AND fbPlasticSorting.bState_HaltDone THEN
					fbStateMachineManual.StateComplete := TRUE;
				END_IF
					
	// =========================================================
	// Turning off axis stop, passing it to axis instances
	E_PMLState.STOPPED:	

				IF bHaltIsSetToTrue THEN
					bHaltIsSetToTrue := FALSE;
					
					fbSeparateModule.Stop(bHalt := FALSE);
					fbMetalSorting.Stop(bHalt := FALSE);
					fbPlasticSorting.Stop(bHalt := FALSE);
				END_IF

				IF fbStateMachineManual.StateComplete THEN
					fbStateMachineManual.StateComplete := FALSE;
				END_IF
				
	// =========================================================
	// Resetting cylinders and axes
	E_PMLState.RESETTING:	

				IF NOT bResetIsSetToTrue THEN
					bResetIsSetToTrue := TRUE;
					
					fbSeparateModule.Reset(bReset := TRUE);							
					fbMetalSorting.Reset(bReset := TRUE);
					fbPlasticSorting.Reset(bReset := TRUE);
				END_IF
				
				IF NOT fbSeparateModule.bState_ResetDone THEN
					fbSeparateModule.Reset(bReset := TRUE);
				END_IF
				
				IF NOT fbMetalSorting.bState_ResetDone THEN
					fbMetalSorting.Reset(bReset := TRUE);
				END_IF
				
				IF NOT fbPlasticSorting.bState_ResetDone THEN
					fbPlasticSorting.Reset(bReset := TRUE);
				END_IF
				
				IF fbSeparateModule.bState_ResetDone AND fbMetalSorting.bState_ResetDone AND fbPlasticSorting.bState_ResetDone 
				AND fbSeparateModule.bState_ClampAtBasePos AND fbSeparateModule.bState_BarrierAtBasePos
				AND fbMetalSorting.bState_CylinderAtBasePos AND fbPlasticSorting.bState_CylinderAtBasePos THEN
					fbStateMachineManual.StateComplete := TRUE;
				END_IF
END_CASE

// =========================================================
END_METHOD

METHOD PRIVATE Operating_Semiautomatic
VAR_INPUT
END_VAR
// =========================================================

CASE ePMLState OF
	
	// =========================================================
	// Turning axis reset off, passing it to axis instances
	E_PMLState.IDLE:		

				IF bResetIsSetToTrue THEN
					bResetIsSetToTrue := FALSE;
					
					fbSeparateModule.Reset(bReset := FALSE);
					fbMetalSorting.Reset(bReset := FALSE);
					fbPlasticSorting.Reset(bReset := FALSE);
					
					fbStateMachineSemiAuto.StateComplete := FALSE;
				END_IF
	
	// =========================================================
	// Resetting variables for executing automatic mode, checking status of axes
	E_PMLState.STARTING:	

				IF NOT bStartingIsSetToTrue THEN
					bStartingIsSetToTrue := TRUE;
					
					fbSeparateModule.Starting(bStarting := TRUE);
					fbMetalSorting.Starting(bStarting := TRUE);
					fbPlasticSorting.Starting(bStarting := TRUE);
				END_IF

				IF NOT fbSeparateModule.bState_StartingDone THEN
					fbSeparateModule.Starting(bStarting := TRUE);
				END_IF
				
				IF NOT fbMetalSorting.bState_StartingDone THEN
					fbMetalSorting.Starting(bStarting := TRUE);
				END_IF
				
				IF NOT fbPlasticSorting.bState_StartingDone THEN
					fbPlasticSorting.Starting(bStarting := TRUE);
				END_IF

				IF fbSeparateModule.bState_StartingDone AND fbMetalSorting.bState_StartingDone AND fbPlasticSorting.bState_StartingDone THEN
					fbStateMachineSemiAuto.StateComplete := TRUE;
				END_IF

	// =========================================================
	// Executing semi-automatic mode
	E_PMLState.EXECUTE:	

				IF bStartingIsSetToTrue THEN
					bStartingIsSetToTrue := FALSE;
					
					fbSeparateModule.Starting(bStarting := FALSE);
					fbMetalSorting.Starting(bStarting := FALSE);
					fbPlasticSorting.Starting(bStarting := FALSE);
					
					fbStateMachineSemiAuto.StateComplete := FALSE;
				END_IF
				
				fbSeparateModule.Semiautomatic();
				fbMetalSorting.Semiautomatic();
				fbPlasticSorting.Semiautomatic();
				
				IF fbTriggerSeparated.Q THEN
					nBoxesOnTheWay := nBoxesOnTheWay + 1;
				END_IF
				
				IF fbTriggerSelectedM.Q THEN
					nBoxesOnTheWay := nBoxesOnTheWay - 1;
				END_IF
				
				IF fbTriggerSelectedP.Q THEN
					nBoxesOnTheWay := nBoxesOnTheWay - 1;
				END_IF
						
	// =========================================================
	// Stopping axes
	E_PMLState.ABORTING:	

				IF NOT bHaltIsSetToTrue THEN
					bHaltIsSetToTrue := TRUE;
	
					fbSeparateModule.Stop(bHalt := TRUE);
					fbMetalSorting.Stop(bHalt := TRUE);
					fbPlasticSorting.Stop(bHalt := TRUE);		
				END_IF

				IF NOT fbSeparateModule.bState_HaltDone THEN
					fbSeparateModule.Stop(bHalt := TRUE);
				END_IF
				
				IF NOT fbMetalSorting.bState_HaltDone THEN
					fbMetalSorting.Stop(bHalt := TRUE);
				END_IF
				
				IF NOT fbPlasticSorting.bState_HaltDone THEN
					fbPlasticSorting.Stop(bHalt := TRUE);
				END_IF

				IF fbSeparateModule.bState_HaltDone AND fbMetalSorting.bState_HaltDone AND fbPlasticSorting.bState_HaltDone THEN
					fbStateMachineSemiAuto.StateComplete := TRUE;
				END_IF
	
	// =========================================================
	// Turning off axis stop, passing it to axis instances
	E_PMLState.ABORTED:	

				IF bHaltIsSetToTrue THEN
					bHaltIsSetToTrue := FALSE;
					
					fbSeparateModule.Stop(bHalt := FALSE);
					fbMetalSorting.Stop(bHalt := FALSE);
					fbPlasticSorting.Stop(bHalt := FALSE);
				END_IF
				
				IF fbStateMachineSemiAuto.StateComplete THEN
					fbStateMachineSemiAuto.StateComplete := FALSE;
				END_IF
	
	// =========================================================
	E_PMLState.CLEARING:	

				fbStateMachineSemiAuto.StateComplete := TRUE;
	
	// =========================================================
	// Selecting boxes on conveyor belt to destination, then stopping axes
	E_PMLState.STOPPING:	

				IF fbTriggerSeparated.Q THEN
					nBoxesOnTheWay := nBoxesOnTheWay + 1;
				END_IF
				
				IF fbTriggerSelectedM.Q THEN
					nBoxesOnTheWay := nBoxesOnTheWay - 1;
				END_IF
				
				IF fbTriggerSelectedP.Q THEN
					nBoxesOnTheWay := nBoxesOnTheWay - 1;
				END_IF
				
				IF (nBoxesOnTheWay = 0) AND NOT bHaltIsSetToTrue THEN
					bHaltIsSetToTrue := TRUE;

					fbSeparateModule.Stop(bHalt := TRUE);
					fbMetalSorting.Stop(bHalt := TRUE);
					fbPlasticSorting.Stop(bHalt := TRUE);						
				END_IF
				
				IF NOT fbSeparateModule.bState_HaltDone OR (nBoxesOnTheWay <> 0) THEN
					fbSeparateModule.Semiautomatic();
					
					IF (nBoxesOnTheWay = 0) THEN
						fbSeparateModule.Stop(bHalt := TRUE);
					END_IF
				END_IF
				
				IF NOT fbMetalSorting.bState_HaltDone OR (nBoxesOnTheWay <> 0) THEN
					fbMetalSorting.Semiautomatic();
					
					IF (nBoxesOnTheWay = 0) THEN
						fbMetalSorting.Stop(bHalt := TRUE);
					END_IF
				END_IF
				
				IF NOT fbPlasticSorting.bState_HaltDone OR (nBoxesOnTheWay <> 0) THEN
					fbPlasticSorting.Semiautomatic();
					
					IF (nBoxesOnTheWay = 0) THEN
						fbPlasticSorting.Stop(bHalt := TRUE);
					END_IF
				END_IF

				IF fbSeparateModule.bState_HaltDone AND fbMetalSorting.bState_HaltDone
				AND fbPlasticSorting.bState_HaltDone AND (nBoxesOnTheWay = 0) THEN
					fbStateMachineSemiAuto.StateComplete := TRUE;
				END_IF
					
	// =========================================================
	// Turning off axis stop, passing it to axis instances
	E_PMLState.STOPPED:	
				
				IF bHaltIsSetToTrue THEN
					bHaltIsSetToTrue := FALSE;
					
					fbSeparateModule.Stop(bHalt := FALSE);
					fbMetalSorting.Stop(bHalt := FALSE);
					fbPlasticSorting.Stop(bHalt := FALSE);
				END_IF
				
				IF fbStateMachineSemiAuto.StateComplete THEN
					fbStateMachineSemiAuto.StateComplete := FALSE;
				END_IF

	// =========================================================
	// Resetting cylinders and axes
	E_PMLState.RESETTING:	

				IF NOT bResetIsSetToTrue THEN
					bResetIsSetToTrue := TRUE;
					
					fbSeparateModule.Reset(bReset := TRUE);							
					fbMetalSorting.Reset(bReset := TRUE);
					fbPlasticSorting.Reset(bReset := TRUE);
				END_IF
				
				IF NOT fbSeparateModule.bState_ResetDone THEN
					fbSeparateModule.Reset(bReset := TRUE);
				END_IF
				
				IF NOT fbMetalSorting.bState_ResetDone THEN
					fbMetalSorting.Reset(bReset := TRUE);
				END_IF
				
				IF NOT fbPlasticSorting.bState_ResetDone THEN
					fbPlasticSorting.Reset(bReset := TRUE);
				END_IF
				
				IF fbSeparateModule.bState_ResetDone AND fbMetalSorting.bState_ResetDone AND fbPlasticSorting.bState_ResetDone 
				AND fbSeparateModule.bState_ClampAtBasePos AND fbSeparateModule.bState_BarrierAtBasePos
				AND fbMetalSorting.bState_CylinderAtBasePos AND fbPlasticSorting.bState_CylinderAtBasePos THEN
					nBoxesOnTheWay 							:= 0;
					fbStateMachineSemiAuto.StateComplete 	:= TRUE;
				END_IF
END_CASE

// =========================================================
END_METHOD

END_FUNCTION_BLOCK

// ---- 02_Subsystems/FB_SeparatingModule.TcPOU
// Module to separate via sensor, barrier and clamp cylinder and axis
FUNCTION_BLOCK FB_SeparatingModule EXTENDS FB_Subsystem_Root
VAR_INPUT
	// =============== Control the state and mode of machine ========================
	bExecute					: BOOL;							// To control the process execution of separating module (true in state EXECUTE)
	bSemiStart					: BOOL;							// To trigger one process exeuction in semi automatic mode
	
	// =============== Information about number of boxes being sorted ===============
	nBoxesOnTheWay				: INT;							// Actual number of boxes being processed
	
	// =============== Cylinders buttons ============================================
	bButtonClampToWorkIn		: BOOL;							// Signal of button to move clamp cylinder to work position
	bButtonClampToBaseIn		: BOOL;							// Signal of button to move clamp cylinder to base position
	bButtonBarrierToWorkIn		: BOOL;							// Signal of button to move barrier cylinder to work position
	bButtonBarrierToBaseIn		: BOOL;							// Signal of button to move barrier cylinder to base position
	
END_VAR
VAR_OUTPUT
	// =============== Process information ==========================================
	bSeparated					: BOOL;							// Gets true if one separating process is done

	// =============== For movement simulation on visualization =====================
	bClampToWork				: BOOL;							// Simulation of clamp cylinder movement to work position
	bBarrierToWork				: BOOL;							// Simulation of barrier cylinder movement to work position
		
	// =============== Error variables ==============================================
	bClampError					: BOOL;							// Error signal of clamp cylinder
	sClampErrorMsg				: STRING;						// Error message of clamp cylinder
	bBarrierError				: BOOL;							// Error signal of barrier cylinder
	sBarrierErrorMsg			: STRING;						// Error message of barrier cylinder
	
	// =============== Temperature recordings =======================================
	aClampTemps					: ARRAY[1..100] OF LREAL;		// Array with recorded temperatures of clamp cylinder
	aBarrierTemps				: ARRAY[1..100] OF LREAL;		// Array with recorded temperatures of barrier cylinder
	
	// =============== Button return signals ========================================
	bButtonClampToWorkOut		: BOOL;							// Processed signal for button to move clamp cylinder to work position
	bButtonClampToBaseOut		: BOOL;							// Processed signal for button to move clamp cylinder to base position
	bButtonBarrierToWorkOut		: BOOL;							// Processed signal for button to move barrier cylinder to work position
	bButtonBarrierToBaseOut		: BOOL;							// Processed signal for button to move barrier cylinder to base position
END_VAR

VAR
	// =============== Function block instance of sensor ============================
	fbSensor					: FB_SignalHandling;			// Sensor needed for separating process
	
	// =============== Function block instances for clamp cylinder ==================
	fbClamp						: FB_Cylinder;					// Without diagnosis and temperature mode
	fbClampDiag					: FB_CylinderDiag;				// With diagnosis of states
	fbClampTemp					: FB_CylinderTemp;				// With temperature mode
	fbClampTempDiag				: FB_CylinderTempDiag;			// With diagnosis of temperature
	fbClampTempRecord			: FB_CylinderTempRecord;		// With record of temperatures
	
	// =============== Interface instance for clamp cylinder ========================
	ipClamp						: I_Cylinder;					// Interface for flexible access to clamp cylinder FBs
	
	// =============== Function block instances for barrier cylinder ================
	fbBarrier					: FB_Cylinder;					// Without diagnosis and temperature mode
	fbBarrierDiag				: FB_CylinderDiag;				// With diagnosis of states
	fbBarrierTemp				: FB_CylinderTemp;				// With temperature mode
	fbBarrierTempDiag			: FB_CylinderTempDiag;			// With diagnosis of temperature
	fbBarrierTempRecord			: FB_CylinderTempRecord;		// With record of temperatures
	
	// =============== Interface instance for barrier cylinder ======================
	ipBarrier					: I_Cylinder;					// Interface for flexible access to barrier cylinder FBs
		
	// =============== Cylinder parameters for clamp and barrier ====================
	tTimeOutClamp				: TIME;							// For clamp cylinder with diagnosis: time in which the cylinder should reach base/work position
	tTimeOutBarrier				: TIME;							// For barrier cylinder with diagnosis: time in which the cylinder should reach base/work position
	tRecordIntervalClamp		: TIME;							// Time of intervals to record the temperature of clamp cylinder
	tRecordIntervalBarrier		: TIME;							// Time of intervals to record the temperature of barrier cylinder
	tBarrierAtWork				: TIME;							// Time value for separating process: barrier cylinder stays at work position
	
	// =============== Manual cylinder control ======================================
	fbButtonClampToWork			: FB_SignalHandlingIntern;		// To move clamp cylinder manually to work position
	fbButtonClampToBase			: FB_SignalHandlingIntern;		// To move clamp cylinder manually to base position
	fbButtonBarrierToWork		: FB_SignalHandlingIntern;		// To move barrier cylinder manually to work position
	fbButtonBarrierToBase		: FB_SignalHandlingIntern;		// To move barrier cylinder manually to base position
	
	// =============== Common variables ==============================================
	fbTimerBarrierAtWork		: TON;							// Timer for opening barrier in (semi) automatic mode
	eStateAuto					: E_StateSeparatingAuto;		// State variable for automatic mode
	eStateSemiAuto				: E_StateSeparatingAuto;		// State variable for semi automatic mode
	
END_VAR

// =========================================================
;
// =========================================================

METHOD Automatic
VAR_INPUT
END_VAR
// =========================================================
// Noticing work position of barrier cylinder	

	fbTimerBarrierAtWork(PT := tBarrierAtWork);

// =========================================================
// Control of main axis

	IF NOT bHaltRequest THEN
		fbAxis.MoveFw();
		
	ELSIF NOT bHaltDone THEN
		Stop(bHalt := TRUE);
		
	ELSE
		Stop(bHalt := FALSE);
	END_IF

// =========================================================
// Process of separating boxes
	
	CASE eStateAuto OF
		
		// =========================================================
		E_StateSeparatingAuto.Init:
		
				// Calling method of FB via interface instance
				ipBarrier.MoveToBase();
				
				// Accessing property of FB via interface instance
				IF ipBarrier.bState_AtBasePos AND bExecute THEN
					eStateAuto := E_StateSeparatingAuto.Start;
				END_IF
			
		// =========================================================
		E_StateSeparatingAuto.Start:
		
				IF fbSensor.bOut AND fbAxis.bMoves THEN
					eStateAuto := E_StateSeparatingAuto.CloseClamp;
				
				// Accessing property of FB via interface instance
				ELSIF NOT ipClamp.bState_AtWorkPos THEN
					// Calling method of FB via interface instance
					ipClamp.MoveToWork();
				END_IF
			
		// =========================================================
		E_StateSeparatingAuto.CloseClamp:
				
				// Calling method of FB via interface instance
				ipClamp.MoveToBase();
				
				// Accessing property of FB via interface instance
				IF ipClamp.bState_AtBasePos THEN
					bSeparated 	:= TRUE;
					eStateAuto 	:= E_StateSeparatingAuto.OpenBarrier;
				END_IF
			
		// =========================================================
		E_StateSeparatingAuto.OpenBarrier:
		
				// Calling method of FB via interface instance
				ipBarrier.MoveToWork();
				
				// Accessing property of FB via interface instance
				IF ipBarrier.bState_AtWorkPos THEN
					fbTimerBarrierAtWork(IN := TRUE);
				END_IF
				
				IF fbTimerBarrierAtWork.Q THEN
					fbTimerBarrierAtWork(IN := FALSE);
					eStateAuto := E_StateSeparatingAuto.CloseBarrier;
				END_IF
			
		// =========================================================
		E_StateSeparatingAuto.CloseBarrier:
		
				// Calling method of FB via interface instance
				ipBarrier.MoveToBase();
				
				// Accessing property of FB via interface instance
				IF ipBarrier.bState_AtBasePos THEN
					bSeparated 	:= FALSE;
					eStateAuto	:= E_StateSeparatingAuto.OpenClamp;
				END_IF
			
		// =========================================================
		E_StateSeparatingAuto.OpenClamp:		
				// Calling method of FB via interface instance
				ipClamp.MoveToWork();
				
				// Accessing property of FB via interface instance
				IF ipClamp.bState_AtWorkPos THEN
					eStateAuto := E_StateSeparatingAuto.Init;
				END_IF
	END_CASE

// =========================================================
END_METHOD

PROPERTY bState_BarrierAtBasePos : BOOL
GET
bState_BarrierAtBasePos := ipBarrier.bState_AtBasePos;
END_GET
END_PROPERTY

PROPERTY bState_BarrierAtWorkPos : BOOL
GET
bState_BarrierAtWorkPos := ipBarrier.bState_AtWorkPos;
END_GET
END_PROPERTY

PROPERTY bState_ClampAtBasePos : BOOL
GET
bState_ClampAtBasePos := ipClamp.bState_AtBasePos;
END_GET
END_PROPERTY

PROPERTY bState_ClampAtWorkPos : BOOL
GET
bState_ClampAtWorkPos := ipClamp.bState_AtWorkPos;
END_GET
END_PROPERTY

METHOD CylinderOptions
VAR_INPUT
	bClampDiag			: BOOL;		// If true the clamp cylinder has diagnosis functionality
	bClampTemp			: BOOL;		// If true the clamp cylinder has temperature functionality
	bClampRecord		: BOOL;		// If true the clamp cylinder has recording functionality
	bBarrierDiag		: BOOL;		// If true the barrier cylinder has diagnosis functionality
	bBarrierTemp		: BOOL;		// If true the barrier cylinder has temperature functionality
	bBarrierRecord		: BOOL;		// If true the barrier cylinder has recording functionality
END_VAR
// =========================================================
// Selecting clamp cylinder

	// Checking variables to enable/disable diagnosis and temperature mode
	IF bClampDiag THEN
		IF bClampTemp THEN
			// ============== FB with diagnosis and temperature mode ==============
			bClampError 	:= fbClampTempDiag.bError;								// Assigning output variable of chosen FB to local output variable
			sClampErrorMsg 	:= fbClampTempDiag.sErrorMsg;
			ipClamp 		:= fbClampTempDiag;										// Assigning chosen FB instance to interface instance
		
		ELSE
			// ============== FB with diagnosis and without temperature mode ==============
			fbClampDiag.tTimeOut 	:= tTimeOutClamp;								// Setting special data for selected FB
			bClampError 			:= fbClampDiag.bError;							// Assigning output variable of chosen FB to local output variable	
			sClampErrorMsg 			:= fbClampDiag.sErrorMsg;
			ipClamp 				:= fbClampDiag;									// Assigning chosen FB instance to interface instance
		END_IF
	ELSE
		bClampError 	:= FALSE;
		sClampErrorMsg 	:= '';
		
		IF bClampTemp THEN
			IF bClampRecord THEN
				// ============== FB without diagnosis and with temperature recording ==============
				fbClampTempRecord.tIntervalTime	:= tRecordIntervalClamp;			// Time of record interval
				fbClampTempRecord.bRecordStart	:= bComprAirEnabledLocal;			// Recording if compressed air is set
				
				fbClampTempRecord.Record();											// Calling method of function block FB_CylinderTempRecord
				
				aClampTemps 	:= fbClampTempRecord.aTemps;						// Saving output variable
				ipClamp 		:= fbClampTempRecord;								// Assigning chosen FB instance to interface instance
			ELSE
				// ============== FB without diagnosis and with temperature mode, but without recording ==============
				ipClamp 		:= fbClampTemp;										// Assigning chosen FB instance to interface instance
			END_IF
		ELSE
			// ============== FB without diagnosis and without temperature mode ==============
			ipClamp := fbClamp;														// Assigning chosen FB instance to interface instance		
		END_IF	
	END_IF
									
// =========================================================
// Selecting barrier cylinder

	// Checking variables to enable/disable diagnosis and temperature mode
	IF bBarrierDiag THEN
		IF bBarrierTemp THEN
			// ============== FB with diagnosis and temperature mode ==============
			bBarrierError 		:= fbBarrierTempDiag.bError;						// Assigning output variable of chosen FB to local output variable
			sBarrierErrorMsg 	:= fbBarrierTempDiag.sErrorMsg;
			ipBarrier 			:= fbBarrierTempDiag;								// Assigning chosen FB instance to interface instance
		
		ELSE
			// ============== FB with diagnosis and without temperature mode ==============
			fbBarrierDiag.tTimeOut	:= tTimeOutBarrier;								// Setting special data for selected FB
			bBarrierError 			:= fbBarrierDiag.bError;						// Assigning output variable of chosen FB to local output variable
			sBarrierErrorMsg 		:= fbBarrierDiag.sErrorMsg;
			ipBarrier 				:= fbBarrierDiag;								// Assigning chosen FB instance to interface instance
		END_IF
	ELSE
		bBarrierError := FALSE;
		sBarrierErrorMsg := '';
		
		IF bBarrierTemp THEN
			IF bBarrierRecord THEN
				// ============== FB without diagnosis and with temperature recording ==============
				fbBarrierTempRecord.tIntervalTime 	:= tRecordIntervalBarrier;		// Time of record interval
				fbBarrierTempRecord.bRecordStart 	:= bComprAirEnabledLocal;		// Recording if compressed air is set
				
				fbBarrierTempRecord.Record();										// Calling method of function block FB_CylinderTempRecord
				
				aBarrierTemps 	:= fbBarrierTempRecord.aTemps;						// Saving output variable
				ipBarrier 		:= fbBarrierTempRecord;								// Assigning chosen FB instance to interface instance
			ELSE
				// ============== FB without diagnosis and with temperature mode, but without recording ==============
				ipBarrier 		:= fbBarrierTemp; 									// Assigning chosen FB instance to interface instance
			END_IF
		ELSE
			// ============== FB without diagnosis and without temperature mode ==============
			ipBarrier := fbBarrier;													// Assigning chosen FB instance to interface instance				
		END_IF	
	END_IF
									
// =========================================================
END_METHOD

METHOD Enable
VAR_INPUT
	bComprAirEnabled		: BOOL;			// Enable of compressed air
	bAxisEnable				: BOOL;			// Enable of axis
	bSensorEnable			: BOOL;			// Enable of sensor
	bManualAxisEnable		: BOOL;			// Enable of manual axis control
END_VAR
// =========================================================
// Calling method Enable of base class FB_Module via 'SUPER^.'
		
	SUPER^.Enable(	bComprAirEnabled	:= bComprAirEnabled,
					bAxisEnable			:= bAxisEnable,
					bSensorEnable		:= bSensorEnable,
					bManualAxisEnable	:= bManualAxisEnable);

// =========================================================
// Sensor control
		
	fbSensor.Enable(bEnable := bSensorEnable);

// =========================================================
// Cylinder control (accessing property of FB via interfaces intances)
	
	// Clamp cylinder
	fbButtonClampToWork.Enable(bEnable := bManualCylinderEnable AND NOT ipClamp.bState_AtWorkPos);		
	fbButtonClampToBase.Enable(bEnable := bManualCylinderEnable AND NOT ipClamp.bState_AtBasePos);
	
	fbButtonClampToBase.bInput 	:= NOT fbButtonClampToWork.bInput;
	
	// Barrier cylinder
	fbButtonBarrierToWork.Enable(bEnable := bManualCylinderEnable AND NOT ipBarrier.bState_AtWorkPos);
	fbButtonBarrierToBase.Enable(bEnable := bManualCylinderEnable AND NOT ipBarrier.bState_AtBasePos);
	
	fbButtonBarrierToBase.bInput := NOT fbButtonBarrierToWork.bInput;

// =========================================================
END_METHOD

METHOD InputOutput
VAR_INPUT
END_VAR
// =========================================================
// Calling method SetOutput of base class FB_Module via 'SUPER^.'
		
	SUPER^.InputOutput();						

// =========================================================
// Sensor
		
	fbSensor.SetOutput();

// =========================================================
// Cylinder buttons
		
	fbButtonClampToWork.SetOutput();
	fbButtonClampToBase.SetOutput();
	fbButtonBarrierToWork.SetOutput();
	fbButtonBarrierToBase.SetOutput();

// =========================================================
// Output variables for cylinders
	
	// Accessing properties of selected FB via interface instances
	bClampToWork 	:= ipClamp.bState_MoveToWork;
	bBarrierToWork 	:= ipBarrier.bState_MoveToWork;

// =========================================================
// Buttons

	fbButtonClampToWork.bInput 		:= bButtonClampToWorkIn;
	fbButtonClampToBase.bInput 		:= bButtonClampToBaseIn;
	fbButtonBarrierToWork.bInput 	:= bButtonBarrierToWorkIn;
	fbButtonBarrierToBase.bInput 	:= bButtonBarrierToBaseIn;
	bButtonClampToWorkOut 			:= fbButtonClampToWork.bOut;
	bButtonClampToBaseOut 			:= fbButtonClampToBase.bOut;
	bButtonBarrierToWorkOut 		:= fbButtonBarrierToWork.bOut;
	bButtonBarrierToBaseOut 		:= fbButtonBarrierToBase.bOut;

// =========================================================
END_METHOD

METHOD Maintenance
VAR_INPUT
END_VAR
// =========================================================
// Calling own method Manual of this class FB_SeparatingModule via 'THIS^.'
		
	THIS^.Manual();				

// =========================================================
END_METHOD

METHOD Manual
VAR_INPUT
END_VAR
// =========================================================
// Calling method Manual of base class FB_Module via 'SUPER^.'
		
	SUPER^.Manual();							

// =========================================================
// Manual cylinder control (Calling methods of FBs via interface instances)
	
	// Clamp cylinder to work position
	IF fbButtonClampToWork.bOut THEN
		ipClamp.MoveToWork();
	// Clamp cylinder to base position
	ELSIF fbButtonClampToBase.bOut THEN
		ipClamp.MoveToBase();
	END_IF
	
	// Barrier cylinder to work position
	IF fbButtonBarrierToWork.bOut THEN
		ipBarrier.MoveToWork();
	// Barrier cylinder to base position
	ELSIF fbButtonBarrierToBase.bOut THEN
		ipBarrier.MoveToBase();
	END_IF

// =========================================================
END_METHOD

METHOD Reset
VAR_INPUT
	bReset		: BOOL;				// True if machine is in state RESETTING
END_VAR
// =========================================================
// Calling method Reset of base class FB_Module via 'SUPER^.'
		
	SUPER^.Reset(bReset := bReset);

// =========================================================
// Resetting cylinder and axis
	
	IF fbTriggerResetStart.Q THEN
		bSeparated := FALSE;
		
		fbTimerBarrierAtWork(IN := FALSE);
		
		// Calling methods of FBs via interface instances
		ipClamp.Reset();
		ipBarrier.Reset();
	END_IF

// =========================================================
END_METHOD

METHOD PROTECTED ResetState
VAR_INPUT
END_VAR
// =========================================================

eStateAuto 		:= E_StateSeparatingAuto.Init;
eStateSemiAuto	:= E_StateSeparatingAuto.Init;

// =========================================================
END_METHOD

METHOD Semiautomatic
VAR_INPUT
END_VAR
// =========================================================
// Noticing work position of barrier cylinder	

	fbTimerBarrierAtWork(PT := tBarrierAtWork);

// =========================================================
// Control of main axis

	IF (nBoxesOnTheWay = 0) AND (eStateSemiAuto = E_StateSeparatingAuto.Init) THEN
		Stop(bHalt := TRUE);
	END_IF
	
	IF bHaltRequest THEN
		IF bHaltDone THEN
			Stop(bHalt := FALSE);
		ELSE
			Stop(bHalt := TRUE);
		END_IF
	ELSE
		fbAxis.MoveFw();
	END_IF

// =========================================================
// Process of separating boxes
	
	CASE eStateSemiAuto OF
		// =========================================================
		E_StateSeparatingAuto.Init:
		
				// Calling method of FB via interface instance
				ipBarrier.MoveToBase();
				
				// Accessing property of FB via interface instance
				IF ipBarrier.bState_AtBasePos AND bExecute AND bSemiStart THEN
					eStateSemiAuto := E_StateSeparatingAuto.Start;
				END_IF
			
		// =========================================================
		E_StateSeparatingAuto.Start:
		
				IF fbSensor.bOut THEN
					eStateSemiAuto := E_StateSeparatingAuto.CloseClamp;
				ELSE
					// Accessing property of FB via interface instance
					IF NOT ipClamp.bState_AtWorkPos THEN
						// Calling method of FB via interface instance
						ipClamp.MoveToWork();
					END_IF
					
					fbAxis.MoveFw();
				END_IF
			
		// =========================================================
		E_StateSeparatingAuto.CloseClamp:
		
				// Calling method of FB via interface instance
				ipClamp.MoveToBase();
				
				// Accessing property of FB via interface instance
				IF ipClamp.bState_AtBasePos THEN
					bSeparated 		:= TRUE;
					eStateSemiAuto 	:= E_StateSeparatingAuto.OpenBarrier;
				END_IF
			
		// =========================================================
		E_StateSeparatingAuto.OpenBarrier:
		
				// Calling method of FB via interface instance
				ipBarrier.MoveToWork();
				
				// Accessing property of FB via interface instance
				IF ipBarrier.bState_AtWorkPos THEN
					fbTimerBarrierAtWork( IN := TRUE );
				END_IF
				
				IF fbTimerBarrierAtWork.Q THEN
					fbTimerBarrierAtWork( IN := FALSE );
					eStateSemiAuto := E_StateSeparatingAuto.CloseBarrier;
				END_IF
			
		// =========================================================
		E_StateSeparatingAuto.CloseBarrier:
		
				// Calling method of FB via interface instance
				ipBarrier.MoveToBase();
				
				// Accessing property of FB via interface instance
				IF ipBarrier.bState_AtBasePos THEN
					bSeparated 		:= FALSE;
					eStateSemiAuto 	:= E_StateSeparatingAuto.OpenClamp;
				END_IF
			
		// =========================================================
		E_StateSeparatingAuto.OpenClamp:
		
				// Calling method of FB via interface instance
				ipClamp.MoveToWork();
				
				// Accessing property of FB via interface instance
				IF ipClamp.bState_AtWorkPos THEN
					eStateSemiAuto := E_StateSeparatingAuto.Init;
				END_IF
	END_CASE

// =========================================================
END_METHOD

PROPERTY tBarrierAtWorkPos : TIME
GET
tBarrierAtWorkPos := tBarrierAtWork;
END_GET
SET
tBarrierAtWork := tBarrierAtWorkPos;
END_SET
END_PROPERTY

PROPERTY tRecordIntervalOfBarrier : TIME
GET
tRecordIntervalOfBarrier := tRecordIntervalBarrier;
END_GET
SET
tRecordIntervalBarrier := tRecordIntervalOfBarrier;
END_SET
END_PROPERTY

PROPERTY tRecordIntervalOfClamp : TIME
GET
tRecordIntervalOfClamp := tRecordIntervalClamp;
END_GET
SET
tRecordIntervalClamp := tRecordIntervalOfClamp;
END_SET
END_PROPERTY

PROPERTY tTimeOutOfBarrier : TIME
GET
tTimeOutOfBarrier := tTimeOutBarrier;
END_GET
SET
tTimeOutBarrier := tTimeOutOfBarrier;
END_SET
END_PROPERTY

PROPERTY tTimeOutOfClamp : TIME
GET
tTimeOutOfClamp := tTimeOutClamp;
END_GET
SET
tTimeOutClamp := tTimeOutOfClamp;
END_SET
END_PROPERTY

END_FUNCTION_BLOCK

// ---- 02_Subsystems/FB_Subsystem_Root.TcPOU
// Base class of modules with axis and buttons for manual control
FUNCTION_BLOCK FB_Subsystem_Root
VAR_INPUT	
	// =============== Axis button variables =====================
	bButtonAxisFwIn				: BOOL;						// Signal of button to move axis forwards
	bButtonAxisBwIn				: BOOL;						// Signal of button to move axis backwards
END_VAR
VAR_OUTPUT
	// =============== Error variables ===========================
	bAxisError					: BOOL;						// Error signal of axis
	nAxisErrorID				: UDINT;					// Error ID of axis error

	// =============== Axis, button and module return signals ====
	bAxisMoves					: BOOL;						// True if axis is moving
	bButtonAxisFwOut			: BOOL;						// Processed signal for button to move axis forwards
	bButtonAxisBwOut			: BOOL;						// Processed signal for button to move axis backwards			
END_VAR
VAR
	// =============== Done signals of Halt, Reset and Starting ==
	bHaltDone					: BOOL;						// True if module is stopped
	bResetDone					: BOOL;						// True if module is reset
	bStartingDone				: BOOL;						// True if module is started
	
	// =============== Enables ===================================
	bComprAirEnabledLocal		: BOOL;						// Enable of compressed air
	bAxisEnableLocal			: BOOL;						// Enable of axis
	bSensorEnableLocal			: BOOL;						// Enable of sensor
	bManualAxisEnableLocal		: BOOL;						// Enable of manual axis control
	bManualCylinderEnable		: BOOL;						// Enable of manual cylinder control (not written with input of method Enable)

	// =============== State variables ===========================
	bHaltRequest				: BOOL;						// True if machine is in state ABORTING or STOPPING
	bResetRequest				: BOOL;						// True if machine is in state RESETTING

	// =============== Axis ======================================
	fbAxis						: FB_Axis;					// Function block instance of FB_Axis
	fAxisVelo					: LREAL;					// Velocity of axis
	
	// =============== Manual axis control =======================
	fbButtonAxisFw				: FB_SignalHandlingIntern;	// To move axis forwards	
	fbButtonAxisBw				: FB_SignalHandlingIntern;	// To move axis backwards
	
	// =============== Common variables ==========================
	fbTriggerStartingStart		: R_TRIG;					// To diagnose rising edge of starting action starting
	fbTriggerResetStart			: R_TRIG;					// To diagnose rising edge of starting reset			
	bMoved						: BOOL;						// History variable to save if axis has moved
END_VAR

// =========================================================
;
// =========================================================

PROPERTY bState_HaltDone : BOOL
GET
bState_HaltDone := bHaltDone;
END_GET
END_PROPERTY

PROPERTY bState_ResetDone : BOOL
GET
bState_ResetDone := bResetDone;
END_GET
END_PROPERTY

PROPERTY bState_StartingDone : BOOL
GET
bState_StartingDone := bStartingDone;
END_GET
END_PROPERTY

METHOD PUBLIC Enable
VAR_INPUT
	bComprAirEnabled		: BOOL;			// Enable of compressed air
	bAxisEnable				: BOOL;			// Enable of axis
	bSensorEnable			: BOOL;			// Enable of sensor
	bManualAxisEnable		: BOOL;			// Enable of manual axis control
END_VAR
// =========================================================
// Store inputs in local variables

	bComprAirEnabledLocal	:= bComprAirEnabled;
	bAxisEnableLocal		:= bAxisEnable;
	bSensorEnableLocal		:= bSensorEnable;
	bManualAxisEnableLocal	:= bManualAxisEnable;
	
// =========================================================	
// Enable axis

	fbAxis.Enable(bEnable := bAxisEnableLocal);					

// =========================================================
// Enable cylinder
		
	bManualCylinderEnable := bManualAxisEnableLocal AND bComprAirEnabledLocal;

// =========================================================
// Control of axis button
		
	fbButtonAxisFw.Enable(bEnable := bManualAxisEnableLocal AND NOT fbButtonAxisBw.bOut);
	fbButtonAxisBw.Enable(bEnable := bManualAxisEnableLocal AND NOT fbButtonAxisFw.bOut);

// =========================================================
END_METHOD

PROPERTY fAxisVelocity : LREAL
GET
fAxisVelocity := fAxisVelo;
END_GET
SET
fAxisVelo := fAxisVelocity;
END_SET
END_PROPERTY

METHOD PUBLIC Halt
VAR_INPUT
	bHalt		: BOOL;				// True if machine is in state ABORTING or STOPPING
END_VAR
// =========================================================
// Store request

	bHaltRequest := bHalt;

// =========================================================
// Halting axis

	fbAxis.Halt(bDriveHalt := bHaltRequest);

// =========================================================
// Getting halt state

	bHaltDone := fbAxis.bState_HaltDone;

// =========================================================
END_METHOD

METHOD PUBLIC InputOutput
VAR_INPUT
END_VAR
// =========================================================
// Axis buttons and output variable for axis
		
	fbButtonAxisFw.SetOutput();	
	fbButtonAxisBw.SetOutput();
	
	bAxisMoves 		:= fbAxis.bMoves;
	bAxisError		:= fbAxis.bError;
	nAxisErrorID	:= fbAxis.nErrorID;
	
	fbButtonAxisFw.bInput 	:= bButtonAxisFwIn;
	fbButtonAxisBw.bInput	:= bButtonAxisBwIn;
	bButtonAxisFwOut 		:= fbButtonAxisFw.bOut;
	bButtonAxisBwOut		:= fbButtonAxisBw.bOut;

// =========================================================
END_METHOD

METHOD PUBLIC Manual
VAR_INPUT
END_VAR
// =========================================================
// Manual axis control
	
	// Button to move axis backwards pressed
	IF fbButtonAxisBw.bOut THEN
		IF bHaltDone THEN
			bHaltDone := FALSE;
		END_IF
		
		IF NOT bMoved THEN
			bMoved := TRUE;
		END_IF
		
		// Move axis backwards
		fbAxis.MoveBw();
	
	// Button to move axis forwards pressed
	ELSIF fbButtonAxisFw.bOut THEN
		IF bHaltDone THEN
			bHaltDone := FALSE;
		END_IF
		
		IF NOT bMoved THEN
			bMoved := TRUE;
		END_IF
		
		// Move axis forwards
		fbAxis.MoveFw();
		
	// No button is pressed and halt is not done
	ELSIF NOT bHaltDone THEN
		// Request halt if axis has moved
		IF bMoved THEN
			Halt(bHalt := TRUE);
		END_IF
		
	// Halt is done but still requested
	ELSIF bHaltRequest THEN
		Halt(bHalt := FALSE);
		
		bMoved := FALSE;
	END_IF

// =========================================================
END_METHOD

METHOD PUBLIC Reset
VAR_INPUT
	bReset		: BOOL;				// True if machine is in state RESETTING
END_VAR
// =========================================================
// Store request

	bResetRequest := bReset;
	
// =========================================================
// Resetting variables

	bMoved 			:= FALSE;
	bHaltDone 		:= FALSE;
	bHaltRequest	:= FALSE;

// =========================================================
// Resetting axis
						
	fbTriggerResetStart(CLK := bReset);
	
	fbAxis.Reset(bDriveReset := bReset);
	
	bResetDone := fbAxis.bState_ResetDone;

// =========================================================
END_METHOD

METHOD PROTECTED ResetState
VAR_INPUT
END_VAR
// =========================================================
// Placeholder method for sub classes
;

// =========================================================
END_METHOD

METHOD PUBLIC Starting
VAR_INPUT
	bStarting		: BOOL;			// True if machine is in state STARTING
END_VAR
// =========================================================

fbTriggerStartingStart(CLK := bStarting);

IF fbTriggerStartingStart.Q THEN
	bStartingDone 			:= FALSE;
	// Setting velocity of axis
	fbAxis.fTargetVelocity 	:= fAxisVelo;
	// Resetting state variable
	ResetState();
END_IF

IF fbAxis.bState_Enable THEN
	bStartingDone := TRUE;
END_IF

// =========================================================
END_METHOD

METHOD PUBLIC Stop
VAR_INPUT
	bHalt		: BOOL;				// True if machine is in state ABORTING or STOPPING
END_VAR
// =========================================================
// Store request

	bHaltRequest := bHalt;

// =========================================================
// Stopping axis

	fbAxis.Stop(bDriveStop := bHaltRequest);
		
// =========================================================			
// Getting halt state

	bHaltDone := fbAxis.bState_HaltDone;

// =========================================================
END_METHOD

END_FUNCTION_BLOCK

// ---- 01_Submodules/Axis/FB_Axis.TcPOU
FUNCTION_BLOCK FB_Axis
VAR_OUTPUT
	// =============== State variables ========================
	bError			: BOOL;					// Error signal
	nErrorID		: UDINT;				// Error ID
	bMoves			: BOOL;					// Status of moving
END_VAR
VAR	
	// =============== Done signals of Halt and Reset =========
	bResetDone		: BOOL;					// Status of function block MC_Reset
	bHaltDone		: BOOL;					// Status of function block MC_Halt

	// =============== State variables ========================
	bStatusEnable	: BOOL;					// Enable feedback
	
	// =============== Velocity, override =====================
	{attribute 'TcAnalytics'}
	fVelocity		: LREAL;				// Target velocity
	fOverride 		: LREAL := 100.0;		// Override 100%
	
	// =============== Trigger function blocks ================
	fbTriggerHalt	: R_TRIG;				// Trigger to recognize rising edge of halt input
	fbTriggerReset	: R_TRIG;				// Trigger to recognize rising edge of reset input
	
	// =============== Axis reference =========================
	AxisRef			: AXIS_REF;				// Axis reference (process data plc/nc)
	
	// =============== Motion function blocks =================
	fbMcPower 		: MC_Power;				// FB for enable and override
	fbMcReset 		: MC_Reset;				// FB to reset axis
	fbMcStop 		: MC_Stop;				// FB to stop axis
	fbMcHalt		: MC_Halt;				// FB to halt axis
	fbMcMove		: MC_MoveVelocity;		// FB to move axis (velocity movement)
END_VAR

// =========================================================
;
// =========================================================

PROPERTY bState_Enable : BOOL
GET
bState_Enable := bStatusEnable;
END_GET
END_PROPERTY

PROPERTY bState_HaltDone : BOOL
GET
bState_HaltDone := bHaltDone;
END_GET
END_PROPERTY

PROPERTY bState_ResetDone : BOOL
GET
bState_ResetDone := bResetDone;
END_GET
END_PROPERTY

METHOD Enable
VAR_INPUT
	bEnable		: BOOL;
END_VAR
// =========================================================

fbMCPower(	Enable 			:= bEnable, 
			Enable_Positive	:= bEnable, 
			Enable_Negative	:= bEnable, 
			Override		:= fOverride,
			Axis			:= AxisRef,
			Status			=> bStatusEnable);
			
IF fbMcPower.Error THEN
	bError		:= TRUE;
	nErrorID 	:= fbMcPower.ErrorID;
END_IF

AxisRef.ReadStatus();

bMoves := AxisRef.Status.Moving;

// =========================================================
END_METHOD

PROPERTY fTargetVelocity : LREAL
GET
fTargetVelocity := fVelocity;
END_GET
SET
fVelocity := fTargetVelocity;
END_SET
END_PROPERTY

METHOD Halt
VAR_INPUT
	bDriveHalt		: BOOL;					// Request stop
END_VAR
// =========================================================

IF bDriveHalt THEN
	// Move Execute FALSE
	fbMCMove(	Execute	:= FALSE,
				Axis 	:= AxisRef);
ELSE
	// Reset done signal
	bHaltDone := FALSE;
END_IF

// Trigger
fbTriggerHalt(CLK := bDriveHalt);

IF fbTriggerHalt.Q THEN
	fbMcHalt(	Execute	:= TRUE,
				Axis 	:= AxisRef);
ELSE
	fbMcHalt(Axis := AxisRef);
END_IF

// Done / Error / Command aborted
IF fbMcHalt.Done OR fbMcHalt.Error OR fbMcHalt.CommandAborted THEN
	bError		:= fbMcHalt.Error;
	nErrorID 	:= fbMcHalt.ErrorID;
	bHaltDone 	:= fbMcHalt.Done;
	
	fbMCMove(	Execute	:= FALSE,
				Axis 	:= AxisRef);
				
	fbMcHalt(	Execute	:= FALSE,
				Axis 	:= AxisRef);
END_IF

// =========================================================
END_METHOD

METHOD MoveBw
VAR_INPUT
END_VAR
// =========================================================

// Not error
IF NOT fbMcMove.Error THEN
	fbMCMove(	Execute 	:= TRUE,
				Velocity 	:= fVelocity,
				Direction 	:= MC_Negative_Direction,
				Axis 		:= AxisRef );
END_IF

// Error / Command aborted
IF fbMCMove.Error OR fbMCMove.CommandAborted THEN
	IF fbMcMove.Error THEN
		bError		:= TRUE;
		nErrorID 	:= fbMCMove.ErrorID;
	END_IF
	
	fbMCMove(	Execute	:= FALSE,
				Axis 	:= AxisRef);
END_IF

// =========================================================
END_METHOD

METHOD MoveFw
VAR_INPUT
END_VAR
// =========================================================

// Not error
IF NOT fbMcMove.Error THEN
	fbMCMove(	Execute 	:= TRUE,
				Velocity 	:= fVelocity,
				Direction 	:= MC_Positive_Direction,
				Axis 		:= AxisRef );
END_IF

// Error / Command aborted
IF fbMCMove.Error OR fbMCMove.CommandAborted THEN
	IF fbMcMove.Error THEN
		bError		:= TRUE;
		nErrorID 	:= fbMCMove.ErrorID;
	END_IF
	
	fbMCMove(	Execute	:= FALSE,
				Axis 	:= AxisRef);
END_IF

// =========================================================
END_METHOD

METHOD Reset
VAR_INPUT
	bDriveReset		: BOOL;					// Request reset
END_VAR
// =========================================================

IF NOT bDriveReset THEN
	bResetDone 	:= FALSE;
END_IF

// Trigger
fbTriggerReset(CLK := bDriveReset);

IF fbTriggerReset.Q THEN
	bHaltDone 	:= FALSE;
	
	fbMcReset(Execute := TRUE, Axis := AxisRef);
ELSE
	fbMcReset(Axis := AxisRef);
END_IF

// Done / Error
IF fbMcReset.Done OR fbMcReset.Error THEN
	bError		:= fbMcReset.Error;
	nErrorID 	:= fbMcReset.ErrorID;
	bResetDone 	:= fbMcReset.Done;

	fbMcReset(	Execute	:= FALSE,
				Axis 	:= AxisRef);
END_IF

// =========================================================
END_METHOD

METHOD Stop
VAR_INPUT
	bDriveStop		: BOOL;					// Request stop
END_VAR
// =========================================================

IF bDriveStop THEN
	// Move Execute FALSE
	fbMCMove(	Execute	:= FALSE,
				Axis 	:= AxisRef);
ELSE
	// Reset done signal
	bHaltDone := FALSE;
END_IF

// Trigger
fbTriggerHalt(CLK := bDriveStop);

IF fbTriggerHalt.Q THEN
	fbMcStop(	Execute	:= TRUE,
				Axis 	:= AxisRef);
ELSE
	fbMcStop(Axis := AxisRef);
END_IF

// Done / Error / Command aborted
IF fbMcStop.Done OR fbMcStop.Error OR fbMcStop.CommandAborted THEN
	bError		:= fbMcStop.Error;
	nErrorID 	:= fbMcStop.ErrorID;
	bHaltDone 	:= fbMcStop.Done;
	
	fbMCMove(	Execute	:= FALSE,
				Axis 	:= AxisRef);
				
	fbMcStop(	Execute	:= FALSE,
				Axis 	:= AxisRef);
END_IF

// =========================================================
END_METHOD

END_FUNCTION_BLOCK

// ---- 01_Submodules/Signal handling/POUs/FB_SignalHandlingIntern.TcPOU
FUNCTION_BLOCK FB_SignalHandlingIntern IMPLEMENTS I_SignalHandling
VAR_INPUT
	bInput				: BOOL;			// Input signal, e.g. sensor signal, enable for fuse
END_VAR
VAR_OUTPUT
	bOut				: BOOL;			// Processed output signal, e.g. delayed, inverted
END_VAR
VAR
	bEnableLocal		: BOOL;			// Enable processing of input signal
END_VAR

// =========================================================
;
// =========================================================

METHOD Enable
VAR_INPUT
	bEnable		: BOOL;
END_VAR
// =========================================================
// Store input in local variable

	bEnableLocal := bEnable;

// =========================================================
END_METHOD

METHOD SetOutput
VAR_INPUT
END_VAR
// =========================================================

bOut := bInput AND bEnableLocal;

// =========================================================
END_METHOD

END_FUNCTION_BLOCK

// ---- 01_Submodules/Signal handling/POUs/FB_SignalHandling.TcPOU
FUNCTION_BLOCK FB_SignalHandling IMPLEMENTS I_SignalHandling
VAR_INPUT
	bInput		AT %I*	: BOOL;			// Hardware input signal, e.g. sensor signal, enable for fuse
END_VAR
VAR_OUTPUT
	bOut		AT %Q* 	: BOOL;			// Processed output signal, e.g. delayed, inverted
END_VAR
VAR
	bEnableLocal		: BOOL;			// Enable processing of input signal
END_VAR

// =========================================================
;
// =========================================================

METHOD Enable
VAR_INPUT
	bEnable		: BOOL;
END_VAR
// =========================================================
// Store input in local variable

	bEnableLocal := bEnable;

// =========================================================
END_METHOD

METHOD SetOutput
VAR_INPUT
END_VAR
// =========================================================
	
bOut := bInput AND bEnableLocal;

// =========================================================
END_METHOD

END_FUNCTION_BLOCK

// ---- 01_Submodules/Cylinder/POUs/FB_Cylinder.TcPOU
(* FB_Cylinder		- number of control signals:
							one direction is controllable
					- type of feedback signal:
							feedback in base and work position		*)
						
